# B&R Automation Studio project ACOPOStrak_DATech_Pilot (part 3)

### Config_1.assembly - 5PC900_TS17_00/mappMotion/TrakOval/Config_1.assembly
```
Element gAsmMain (Type=assembly)
  Tracks:
    TrackSeparation = 0.030
    Track[1]:
      Segments:
        SegmentRef[1] = ::Seg_A_1
        SegmentRef[2] = ::Seg_A_2
        SegmentRef[3] = ::Seg_A_3
        SegmentRef[4] = ::Seg_A_4
        SegmentRef[5] = ::Seg_A_5
        SegmentRef[6] = ::Seg_A_6
        SegmentRef[7] = ::Seg_A_7
        SegmentRef[8] = ::Seg_A_8
        SegmentRef[9] = ::Seg_A_9
        SegmentRef[10] = ::Seg_A_10
        SegmentRef[11] = ::Seg_A_11
        SegmentRef[12] = ::Seg_A_12
        SegmentRef[13] = ::Seg_A_13
        SegmentRef[14] = ::Seg_A_14
        SegmentRef[15] = ::Seg_A_15
        SegmentRef[16] = ::Seg_A_16
        SegmentRef[17] = ::Seg_A_17
        SegmentRef[18] = ::Seg_A_18
        SegmentRef[19] = ::Seg_A_19
        SegmentRef[20] = ::Seg_A_20
        SegmentRef[21] = ::Seg_A_21
        SegmentRef[22] = ::Seg_A_22
        SegmentRef[23] = ::Seg_A_23
        SegmentRef[24] = ::Seg_A_24
        SegmentRef[25] = ::Seg_A_25
        SegmentRef[26] = ::Seg_A_26
      Position = Absolute
        SegmentRef = ::Seg_A_11
        SegmentCountDirection = RightToLeft
        Position = 0
        Translation:
          X = 0.0
          Y = 0.0
          Z = 0.0
        Orientation:
          Angle1 = 0.0
          Angle2 = 0.0
          Angle3 = 180
  CommonSegmentSettings:
    SegmentSimulationOnPLC = Off
    ElongationCompensation = Inactive
    StopReaction = InductionHalt
    SpeedFilter = Lowpass
      FilterTime = 0.002
    ControllerParameters:
      DefaultParameter:
        Controller:
          Position:
            ProportionalGain = 220
          Speed:
            ProportionalGain = 60
            IntegrationTime = 0.0
          FeedForward:
            TotalMass = 1.8
            ForcePositive = 2
            ForceNegative = 2
            SpeedForceFactor = 2
            ForceLoad = 0.0
        MovementErrorLimits:
          PositionError = 1
          VelocityError = 100
      AdditionalParameterSets = NotUsed
    ScopeOfErrorReaction = Assembly
    ShuttleIdentificationTime = 2
  Shuttles:
    MaxShuttleCount = 50
    DistanceReserve:
      Collision = 0.002
      ErrorStop = 0.006
    ShuttleStereotypes:
      ShuttleStRef[1] = ShuttleStereotype_1
    MagnetPlateConfigurations:
      ShuttleType[1] = 8F1SA.203.xxxxxx-x
    CollisionAvoidance:
      Strategy = Constant
      MaximumModelDimensions:
        Length:
          ExtentToFront = 0.07
          ExtentToBack = 0.07
        Width:
          Width = 0.046
  AssemblyFeatures:
    AssemblyFeatureRef[1] = gSecLimit
    AssemblyFeatureRef[2] = Feature_Sim_Shuttle_Def
  Visualization:
    MonitoringPv = gShuttleMon
    ProcessingTaskClass = 1
```

### Config_2.shuttlestereotype - 5PC900_TS17_00/mappMotion/TrakOval/Config_2.shuttlestereotype
```
Element ShuttleStereotype_1 (Type=shuttlestereotype)
  MeasurementUnit = 5067858
  MeasurementResolution = 0.00001
  MovementLimits = Internal
    VelocityIsReadOnly = 0
    Velocity:
      Velocity = 2.5
    AccelerationIsReadOnly = 0
    Acceleration:
      Acceleration = 25
    DecelerationIsReadOnly = 0
    Deceleration:
      Deceleration = 25
    UpdateMode = Immediately
  JerkFilter = Used
    JerkTime = 0.02
  UserData:
    Size = 64
```

### Config_3.sector - 5PC900_TS17_00/mappMotion/TrakOval/Config_3.sector
```
Element SectorTrackA_1 (Type=sector)
  Type = Composed
    StartSegment:
      SegmentRef = ::Seg_A_24
    EndSegment:
      SegmentRef = ::Seg_A_25
      Position = 0
      PositionRelativeTo = FromEnd
Element SectorTrackA_2 (Type=sector)
  Type = Composed
    StartSegment:
      SegmentRef = ::Seg_A_3
    IntermediateSegments:
      SegmentRef[1] = ::Seg_A_4
      SegmentRef[2] = ::Seg_A_5
      SegmentRef[3] = ::Seg_A_6
    EndSegment:
      SegmentRef = ::Seg_A_7
      PositionRelativeTo = FromEnd
Element SectorTrackA_3 (Type=sector)
  Type = Composed
    StartSegment:
      SegmentRef = ::Seg_A_11
    EndSegment:
      SegmentRef = ::Seg_A_12
      PositionRelativeTo = FromEnd
Element SectorTrackA_4 (Type=sector)
  Type = Composed
    StartSegment:
      SegmentRef = ::Seg_A_16
    IntermediateSegments:
      SegmentRef[1] = ::Seg_A_17
      SegmentRef[2] = ::Seg_A_18
      SegmentRef[3] = ::Seg_A_19
    EndSegment:
      SegmentRef = ::Seg_A_20
      PositionRelativeTo = FromEnd
Element SectorTrackAll (Type=sector)
  Type = Composed
    StartSegment:
      SegmentRef = ::Seg_A_26
    IntermediateSegments:
      SegmentRef[1] = ::Seg_A_1
      SegmentRef[2] = ::Seg_A_2
      SegmentRef[3] = ::Seg_A_3
      SegmentRef[4] = ::Seg_A_4
      SegmentRef[5] = ::Seg_A_5
      SegmentRef[6] = ::Seg_A_6
      SegmentRef[7] = ::Seg_A_7
      SegmentRef[8] = ::Seg_A_8
      SegmentRef[9] = ::Seg_A_9
      SegmentRef[10] = ::Seg_A_10
      SegmentRef[11] = ::Seg_A_11
      SegmentRef[12] = ::Seg_A_12
      SegmentRef[13] = ::Seg_A_13
      SegmentRef[14] = ::Seg_A_14
      SegmentRef[15] = ::Seg_A_15
      SegmentRef[16] = ::Seg_A_16
      SegmentRef[17] = ::Seg_A_17
      SegmentRef[18] = ::Seg_A_18
      SegmentRef[19] = ::Seg_A_19
      SegmentRef[20] = ::Seg_A_20
      SegmentRef[21] = ::Seg_A_21
      SegmentRef[22] = ::Seg_A_22
      SegmentRef[23] = ::Seg_A_23
      SegmentRef[24] = ::Seg_A_24
    EndSegment:
      SegmentRef = ::Seg_A_25
      PositionRelativeTo = FromEnd
Element Sector3D (Type=sector)
  Type = Composed
    StartSegment:
      SegmentRef = ::Seg_A_19
      Position = 0.22
    EndSegment:
      SegmentRef = ::Seg_A_19
      Position = 0
      PositionRelativeTo = FromEnd
Element SectorCurve1 (Type=sector)
  Type = Composed
    StartSegment:
      SegmentRef = ::Seg_A_26
    IntermediateSegments:
      SegmentRef[1] = ::Seg_A_1
    EndSegment:
      SegmentRef = ::Seg_A_2
      PositionRelativeTo = FromEnd
Element SectorCurve2 (Type=sector)
  Type = Composed
    StartSegment:
      SegmentRef = ::Seg_A_19
    IntermediateSegments:
      SegmentRef[1] = 
    EndSegment:
      SegmentRef = ::Seg_A_19
      PositionRelativeTo = FromEnd
Element SectorCurve3 (Type=sector)
  Type = Composed
    StartSegment:
      SegmentRef = ::Seg_A_13
    IntermediateSegments:
      SegmentRef[1] = ::Seg_A_14
    EndSegment:
      SegmentRef = ::Seg_A_15
      PositionRelativeTo = FromEnd
Element SectorCurve4 (Type=sector)
  Type = Composed
    StartSegment:
      SegmentRef = ::Seg_A_21
    IntermediateSegments:
      SegmentRef[1] = ::Seg_A_22
    EndSegment:
      SegmentRef = ::Seg_A_23
      PositionRelativeTo = FromEnd
```

### Config_4.processpointlist - 5PC900_TS17_00/mappMotion/TrakOval/Config_4.processpointlist
```
Element ProcessPointList_1 (Type=processpointlist)
  ProcessPoint[0]:
    Name = ptCheckOut
    SectorRef = SectorTrackAll
    Position = 0.1
    PositionRelativeTo = FromEnd
    TriggerEventBufferSize = 10
    BarrierFunctionality = On
  ProcessPoint[1]:
    Name = ptCheckIn
    SectorRef = SectorTrackAll
    Position = 0.66
    PositionRelativeTo = FromEnd
    TriggerEventBufferSize = 30
    BarrierFunctionality = On
  ProcessPoint[2]:
    Name = pt3DIn
    SectorRef = SectorTrackAll
    Position = 10.52
    TriggerEventBufferSize = 10
    BarrierFunctionality = Off
  ProcessPoint[3]:
    Name = pt3DOut
    SectorRef = SectorTrackAll
    Position = 10.588
    PositionRelativeTo = FromEnd
    TriggerEventBufferSize = 10
    BarrierFunctionality = Off
  ProcessPoint[4]:
    Name = pt3D
    SectorRef = Sector3D
    TriggerEventBufferSize = 10
    BarrierFunctionality = Off
  ProcessPoint[5]:
    Name = ptCSZInt
    SectorRef = SectorTrackA_4
    Position = 1.76
    TriggerEventBufferSize = 10
    BarrierFunctionality = On
  ProcessPoint[6]:
    Name = ptCSZIn
    SectorRef = SectorTrackA_4
    Position = 1.75
    TriggerEventBufferSize = 10
    BarrierFunctionality = On
  ProcessPoint[7]:
    Name = ptCSZOut
    SectorRef = SectorTrackA_4
    Position = 2.02
    TriggerEventBufferSize = 10
    BarrierFunctionality = On
  ProcessPoint[8]:
    Name = ptUnloadingIn
    SectorRef = SectorCurve4
    Position = 0.76
    TriggerEventBufferSize = 10
    BarrierFunctionality = On
  ProcessPoint[9]:
    Name = ptUnloadingOut
    SectorRef = SectorCurve4
    Position = 0.88
    TriggerEventBufferSize = 10
    BarrierFunctionality = On
  ProcessPoint[10]:
    Name = ptVision
    SectorRef = SectorTrackAll
    Position = 7.1
    TriggerEventBufferSize = 10
    BarrierFunctionality = On
Element ProcessPointList_2 (Type=processpointlist)
  ProcessPoint[0]:
    Name = ptStage1
    SectorRef = SectorCurve1
    Position = 0.2295
    TriggerEventBufferSize = 10
    BarrierFunctionality = Off
  ProcessPoint[1]:
    Name = ptStage2
    SectorRef = SectorTrackA_2
    Position = 0.1778
    TriggerEventBufferSize = 10
    BarrierFunctionality = Off
  ProcessPoint[2]:
    Name = ptStage3
    SectorRef = SectorTrackA_2
    Position = 0.482
    TriggerEventBufferSize = 10
    BarrierFunctionality = Off
  ProcessPoint[3]:
    Name = ptStage4
    SectorRef = SectorTrackA_2
    Position = 0.715
    TriggerEventBufferSize = 10
    BarrierFunctionality = Off
  ProcessPoint[4]:
    Name = ptStage5
    SectorRef = SectorTrackA_2
    Position = 0.9375
    TriggerEventBufferSize = 10
    BarrierFunctionality = Off
  ProcessPoint[5]:
    Name = ptStage6
    SectorRef = SectorTrackA_2
    Position = 1.036
    TriggerEventBufferSize = 10
    BarrierFunctionality = Off
  ProcessPoint[6]:
    Name = ptStage7
    SectorRef = SectorTrackA_2
    Position = 2.231
    TriggerEventBufferSize = 10
    BarrierFunctionality = Off
  ProcessPoint[7]:
    Name = ptStage8
    SectorRef = SectorTrackA_2
    Position = 2.6712
    TriggerEventBufferSize = 10
    BarrierFunctionality = Off
  ProcessPoint[8]:
    Name = ptStage9
    SectorRef = SectorTrackA_2
    Position = 3.151
    TriggerEventBufferSize = 10
    BarrierFunctionality = Off
  ProcessPoint[9]:
    Name = ptStage10
    SectorRef = SectorTrackA_3
    Position = 0.801
    TriggerEventBufferSize = 10
    BarrierFunctionality = Off
  ProcessPoint[10]:
    Name = ptStage11
    SectorRef = SectorCurve3
    Position = 1.1005
    TriggerEventBufferSize = 10
    BarrierFunctionality = Off
  ProcessPoint[11]:
    Name = ptStage12
    SectorRef = SectorTrackA_4
    Position = 0.3805
    TriggerEventBufferSize = 10
    BarrierFunctionality = Off
  ProcessPoint[12]:
    Name = ptStage13
    SectorRef = SectorTrackA_4
    Position = 1.0407
    TriggerEventBufferSize = 10
    BarrierFunctionality = Off
  ProcessPoint[13]:
    Name = ptStage14
    SectorRef = SectorTrackA_4
    Position = 2.0096
    TriggerEventBufferSize = 10
    BarrierFunctionality = Off
  ProcessPoint[14]:
    Name = ptStage15
    SectorRef = SectorTrackA_4
    Position = 2.751
    TriggerEventBufferSize = 10
    BarrierFunctionality = Off
  ProcessPoint[15]:
    Name = ptStage16
    SectorRef = SectorTrackA_4
    Position = 2.8605
    TriggerEventBufferSize = 10
    BarrierFunctionality = Off
  ProcessPoint[16]:
    Name = ptStage17
    SectorRef = SectorCurve4
    Position = 0.121
    TriggerEventBufferSize = 10
    BarrierFunctionality = Off
  ProcessPoint[17]:
    Name = ptStage18
    SectorRef = SectorCurve4
    Position = 0.9179
    TriggerEventBufferSize = 10
    BarrierFunctionality = Off
  ProcessPoint[18]:
    Name = ptStage19
    SectorRef = SectorTrackA_1
    Position = 0.601
    TriggerEventBufferSize = 10
    BarrierFunctionality = Off
  ProcessPoint[19]:
    Name = ptBuffer
    SectorRef = SectorTrackAll
    Position = 0
    TriggerEventBufferSize = 10
    BarrierFunctionality = On
```

### Limits.assemblyfeature - 5PC900_TS17_00/mappMotion/TrakOval/Limits.assemblyfeature
```
Element gSecLimit (Type=assemblyfeature)
  Type = LocalLimits
    LocalLimit[1]:
      Location:
        SectorRef = Sector3D
      MotionLimits:
        Velocity = Basic
          Velocity = 0.25
```

### cfgAudit.mpaudittrail - 5PC900_TS17_00/mappServices/cfgAudit.mpaudittrail
```
Element gAuditTrak (Type=mpaudittrail)
  Audit:
    Events:
      [0] = 18
    RecordingSize = 16384
    SramBufferSize = 128
    TextSource = TXT
      OutputFormat = MpAudit/Event/Root
      Display = Ne
        Format = MpAudit/Event/RootDis
    Export:
      Encrypt = FALSE
  Alarms = None
```

### viCompCR.visioncomponent - 5PC900_TS17_00/mappVision/viCompCR.visioncomponent
```
Element gCameraCodeReading (Type=visioncomponent)
  VisionApplicationReference = ViAppCodeReading
```

## Logical view

Binary libraries used (declarations not repeated): operator, runtime, astime, AsIecCon, AsBrStr, standard, sys_lib, AsIODiag, McBase, McAcpTrak, McAxis, ViBase 5.15.0, AsZip, FileIO, AsARCfg, powerlnk, AsEPL, AsIO, CoTrace, MpAxis, MpBase, McAcpAx, MTTypes, MTBasics 2.00.0, MTData 2.00.0, MTFilter 2.00.0, brsystem, AsBrMath, AsMbTCP, MpAudit 5.15.0

### Global.typ - Global data types
```iecst
(**)

TYPE
	E_ASM_STATUS :
		(
		E_ASM_UNKNOWN := 0,
		E_ASM_OFF := 1,
		E_ASM_ON := 2,
		E_ASM_IDLE := 3,
		E_ASM_PROCESS := 4,
		E_ASM_ERRORSTOP := 5,
		E_ASM_MANUAL := 6,
		E_ASM_POWER_ON := 10,
		E_ASM_POWER_OFF := 20,
		E_ASM_INITIALIZATION := 30,
		E_ASM_RECOVERY := 31,
		E_ASM_RESET := 40,
		E_ASM_STOPPING := 50,
		E_ASM_EMS := 60,
		E_ASM_CLEAN := 70
		);
	E_PROCESS_STATUS :
		(
		E_PROCESS_None,
		E_PROCESS_Stage1,
		E_PROCESS_Stage2,
		E_PROCESS_Stage3,
		E_PROCESS_Stage4,
		E_PROCESS_Stage5,
		E_PROCESS_Stage6,
		E_PROCESS_Stage7,
		E_PROCESS_Stage8,
		E_PROCESS_Stage9,
		E_PROCESS_Stage10,
		E_PROCESS_Stage11,
		E_PROCESS_Stage12,
		E_PROCESS_Stage13,
		E_PROCESS_Stage14,
		E_PROCESS_Stage15,
		E_PROCESS_Stage16,
		E_PROCESS_Stage17,
		E_PROCESS_Stage18,
		E_PROCESS_Stage19
		);
END_TYPE

(**)

TYPE
	ShuttleUserData_typ : 	STRUCT
		SerialNumber : STRING[19]; (*Shuttle Number*)
		ProcessStatus : E_PROCESS_STATUS;
		Data : ARRAY[0..19]OF UINT;
	END_STRUCT;
END_TYPE

(**)

TYPE
	Command_type : 	STRUCT
		PowerOn : BOOL;
		PowerOff : BOOL;
		Initialize : BOOL;
		EMS : BOOL;
		Start : BOOL;
		Stop : BOOL;
		Reset : BOOL;
		ErrorReset : BOOL;
		Clean : BOOL;
	END_STRUCT;
	Parameter_type : 	STRUCT
		MovementPar : MovementParameter_type;
		PositionOffset : PosOffsetParameter_type;
		ProcessPosition : PositionParameter_type;
		TargetPPM : UINT := 30;
		CountOfGroup : USINT := 6;
	END_STRUCT;
	Status_type : 	STRUCT
		AsmState : E_ASM_STATUS;
	END_STRUCT;
END_TYPE

(**)

TYPE
	MovementParameter_type : 	STRUCT
		Initialize : SerializeParType;
		Stage1 : ServeStageParType;
		Stage2 : TransferStageParType;
		Stage3 : TransferStageParType;
		Stage4 : TransferStageParType;
		Stage5 : TransferStageParType;
		Stage6 : TransferStageParType;
		Stage7 : TransferStageParType;
		Stage8 : TransferStageParType;
		Stage9 : TransferStageParType;
		Stage10 : TransferStageParType;
		Stage11 : TransferStageParType;
		Stage12 : TransferStageParType;
		Stage13 : TransferStageParType;
		Stage14 : TransferStageParType;
		Stage15 : TransferStageParType;
		Stage16 : TransferStageParType;
		Stage17 : TransferStageParType;
		Stage18 : TransferStageParType;
		Stage19 : TransferStageParType;
		Return : SerializeParType;
	END_STRUCT;
	PositionParameter_type : 	STRUCT
		Stage : ARRAY[0..18]OF LREAL;
	END_STRUCT;
	PosOffsetParameter_type : 	STRUCT
		Stage : ARRAY[0..18]OF LREAL;
	END_STRUCT;
END_TYPE

(**)

TYPE
	ServeStageParType : 	STRUCT
		Velocity : REAL;
		Acceleration : REAL;
		Deceleration : REAL;
		MaxController : USINT;
	END_STRUCT;
	TransferStageParType : 	STRUCT
		Velocity : REAL;
		Acceleration : REAL;
		Deceleration : REAL;
		MaxController : USINT;
	END_STRUCT;
	SerializeParType : 	STRUCT
		RoutedVelocity : REAL;
		Velocity : REAL;
		Acceleration : REAL;
		Deceleration : REAL;
	END_STRUCT;
END_TYPE

(**)
```

### Global.var - Global variables
```iecst
VAR
	gShuttleMon : McAcpTrakAssemblyMonData;
END_VAR
(**)
VAR
	gLocal : BOOL;
	gManual : BOOL;
	gCmdRemote : Command_type;
	gCmd : Command_type;
END_VAR
VAR RETAIN
	gParInitialized : BOOL;
	gPar : Parameter_type;
END_VAR
VAR
	gSts : Status_type;
END_VAR
(**)
VAR
	gSim : BOOL;
END_VAR
(**)
VAR
	SIZE_OF_USERDATA : UDINT := 64; (*24*)
END_VAR
(*3D *)
VAR
	g3DStartPos : LREAL := 10.52;
	g3DEndPos : LREAL := 10.588;
END_VAR
(*Vision*)
VAR
	gShuttleTotalCount : DINT;
	gInitialDone : BOOL;
END_VAR
(*Barrier at buffer*)
VAR
	BrBuffer : MC_BR_BarrierCommand_AcpTrak;
END_VAR
```

### GlobalConst.var
```iecst
VAR CONSTANT
	ASM_MAX_TARGET : USINT := 20;
END_VAR
```

### Package Logical/Libraries - Global libraries

### Library Logical/Libraries/MyTrak (ANSIC)
Depends on: standard, AsBrStr, McAcpTrak, McAxis, McBase

#### Types.typ
```iecst
(**)
(*Enumeration*)

TYPE
	E_SLOT_IF_STATE :
		(
		E_SLOT_UNKNOWN := 0,
		E_SLOT_MANUAL := 1,
		E_SLOT_IDLE := 2,
		E_SLOT_PROCESS_READY := 3,
		E_SLOT_PROCESSING := 4,
		E_SLOT_TAKEOUT_READY := 5
		) := E_SLOT_UNKNOWN;
END_TYPE

(**)
(*Structure*)

TYPE
	MyTrakSlotType : 	STRUCT  (*Slot of Stage.*)
		Enable : BOOL;
		Sector : UDINT;
		Position : LREAL;
		Interface : E_SLOT_IF_STATE;
		Shuttle : McAxisType;
		NextStage : UDINT;
	END_STRUCT;
	MyTrakSlotTransType : 	STRUCT  (*Function Block for transfer Shuttle from Prestage to Nextstage*)
		moveAbs : MC_BR_RoutedMoveAbs_AcpTrak;
		axis : McAxisType;
		targetSlot : REFERENCE TO MyTrakSlotType;
		next : REFERENCE TO MyTrakSlotTransType;
	END_STRUCT;
	MyTrakSerializeType : 	STRUCT  (*Function Block for transfer Shuttle from Prestage to Nextstage*)
		moveVel : MC_BR_RoutedMoveVel_AcpTrak;
		axis : McAxisType;
		sourceSlot : REFERENCE TO MyTrakSlotType;
		next : REFERENCE TO MyTrakSerializeType;
	END_STRUCT;
END_TYPE

(**)
(*Internal Structrue for FunctionBlock*)

TYPE
	MyTrak_ServeStage_Internal_type : 	STRUCT
		slotMoveFc : REFERENCE TO MyTrakSlotTransType;
		fbTrgInfo : MC_BR_TrgPointGetInfo_AcpTrak;
		fbTrgEnable : MC_BR_TrgPointEnable_AcpTrak;
	END_STRUCT;
	MyTrak_TransStage_Internal_type : 	STRUCT
		slotMoveFc : REFERENCE TO MyTrakSlotTransType;
		manualCmd : R_TRIG;
	END_STRUCT;
	MyTrak_Serialize_Internal_type : 	STRUCT
		serialMoveFc : REFERENCE TO MyTrakSerializeType;
		manualCmd : R_TRIG;
	END_STRUCT;
	MyTrak_TicketArea_Internal_type : 	STRUCT
		step : USINT;
		init : BOOL;
		fbInEnable : MC_BR_TrgPointEnable_AcpTrak;
		fbInGetInfo : MC_BR_TrgPointGetInfo_AcpTrak;
		fbBarrierReadInfo : MC_BR_BarrierReadInfo_AcpTrak;
		fbBarrier : MC_BR_BarrierCommand_AcpTrak;
		fbOutEnable : MC_BR_TrgPointEnable_AcpTrak;
		fbOutGetInfo : MC_BR_TrgPointGetInfo_AcpTrak;
	END_STRUCT;
	MyTrak_ChangeVel_Internal_type : 	STRUCT
		step : DINT;
		preActive : BOOL;
		ElasticMoveVel : MC_BR_ElasticMoveVel_AcpTrak;
		TrgEnable : MC_BR_TrgPointEnable_AcpTrak;
		TrgGetInfo : MC_BR_TrgPointGetInfo_AcpTrak;
	END_STRUCT;
	MyTrak_ShInfeeder_Internal_type : 	STRUCT
		BarCmd : MC_BR_BarrierCommand_AcpTrak;
		BarReadInfo : MC_BR_BarrierReadInfo_AcpTrak;
		Tmr : TON;
		manualCmd : R_TRIG;
	END_STRUCT;
	MyTrak_Buffer_Internal_type : 	STRUCT
		slotMoveFc : REFERENCE TO MyTrakSlotTransType;
		CheckInPointEnable : MC_BR_TrgPointEnable_AcpTrak;
		GetCheckInShuttleInfo : MC_BR_TrgPointGetInfo_AcpTrak;
		GetShuttleInfo : MC_BR_ShReadInfo_AcpTrak;
		CheckOutBarrier : MC_BR_BarrierCommand_AcpTrak;
		Tmr : TON;
		manualCmd : R_TRIG;
		outReqCount : USINT;
	END_STRUCT;
	MyTrak_UntilStop_Internal_type : 	STRUCT
		serialMoveFc : REFERENCE TO MyTrakSerializeType;
		getShuttle : MC_BR_SecGetShuttleSel_AcpTrak;
	END_STRUCT;
END_TYPE
```

#### Constants.var
```iecst
(**)
VAR CONSTANT
	MyTrakIdle : DINT := 0;
	MyTrakRun : DINT := 1;
	MyTrakManual : DINT := 2;
	MyTrakNotEnoughShuttle : DINT := 40000;
	MyTrakMaximumControllerOverflow : DINT := 40001;
	MyTrakMinimumControllerUnderflow : DINT := 40002;
	MyTrakBusy : DINT := 65534;
	MyTrakDisabled : DINT := 65535;
END_VAR
(**)
VAR CONSTANT
	MyTrakNotExistSourceStage : DINT := -40000;
	MyTrakNotExistTargetStage : DINT := -40001;
	MyTrakNotExistSourceProcessPoint : DINT := -40002;
	MyTrakNotExistSourceCheckIn : DINT := -40003;
	MyTrakNotExistSourceCheckOut : DINT := -40004;
	MyTrakNotExistCheckinPt : DINT := -40000;
END_VAR
```

#### MyTrak.fun - Function and Function Block Define
```iecst
(**)
(*Function Blocks*)

{REDUND_ERROR} FUNCTION_BLOCK MyTrak_ShInfeeder (*Buffer Handle based Productivity *) (*$GROUP=User,$CAT=User,$GROUPICON=User.png,$CATICON=User.png*)
	VAR_INPUT
		Enable : BOOL; (*Enable/Disable*)
		ProcessPoint : REFERENCE TO McProcessPointType; (*Stop Position Process Point*)
		SetPPM : UINT; (*SettedPPM*)
		CountOfOneShot : USINT; (*Supply Shuttle Count at once*)
		Process : BOOL; (*Feeding Start/Stop*)
		Pause : BOOL; (*Puase when feeding is started*)
		Manual : BOOL; (*Manual Input when Feeding is Stopped - Positive Trigger*)
	END_VAR
	VAR_OUTPUT
		Active : BOOL; (*Activated FunctionBlock*)
		Error : BOOL; (*Error Status - Not Implemented*)
		ErrorID : DINT; (*Function Block Status - refer to Constant*)
		ActPPM : UINT; (*Actual PPM*)
		Interval : REAL; (*Feeding Interval*)
	END_VAR
	VAR
		Internal : MyTrak_ShInfeeder_Internal_type;
	END_VAR
END_FUNCTION_BLOCK

{REDUND_ERROR} FUNCTION_BLOCK MyTrak_Buffer (*Buffer Handing based Productivity*) (*$GROUP=User,$CAT=User,$GROUPICON=User.png,$CATICON=User.png*)
	VAR_INPUT
		Enable : BOOL; (*Activate Function Block*)
		CheckInProcessPoint : REFERENCE TO McProcessPointType; (*Check In Process Point*)
		CheckOutProcessPoint : REFERENCE TO McProcessPointType; (*Check Out Process Point*)
		TargetStage : UDINT; (*Reference of Target Stage(MyTrakSlotType array)*)
		TargetSlotCount : USINT; (*Count of slot in target stage*)
		Process : BOOL; (*Process Start And Stop*)
		Feeding : BOOL; (*Holding Process*)
		Manual : BOOL; (*Manual Feeding*)
		SetPPM : UINT; (*Set PPM*)
		CountOfOneShot : USINT; (*Feeding Shuttle Count of One Time*)
		MaximumShuttleCount : USINT; (*Maximum Handle Shuttle Count*)
		Velocity : REAL; (*Velocity from Buffer to 'Target Stage'*)
		Acceleration : REAL; (*Acceleration from Buffer to 'Target Stage'*)
		Deceleration : REAL; (*Deceleration from Buffer to 'Target Stage'*)
		AdvancedParameters : McAcpTrakAdvRouteParType; (*Advanced Parameter*)
	END_VAR
	VAR_OUTPUT
		Active : BOOL; (*Activate Status*)
		Error : BOOL; (*Error Status*)
		ErrorID : DINT; (*Error ID*)
		CountOfShuttle : USINT; (*Total Shuttle by Handled By this FunctionBlock*)
		CountOfBuffer : USINT; (*Shuttle Count in Buffer*)
		CountOfSupplied : UDINT; (*Shuttle Count in Buffer*)
		NextSlotNo : INT; (*Next Slot Number*)
		Interval : REAL; (*Feeding Interval*)
	END_VAR
	VAR
		Internal : MyTrak_Buffer_Internal_type;
	END_VAR
END_FUNCTION_BLOCK

{REDUND_ERROR} FUNCTION_BLOCK MyTrak_ServeStage (*Move shuttles  from source process point to stage*) (*$GROUP=User,$CAT=User,$GROUPICON=User.png,$CATICON=User.png*)
	VAR_INPUT
		Enable : BOOL; (*Activate Function Block*)
		SourceProcessPoint : REFERENCE TO McProcessPointType; (*Reference of Process Point that shuttle getting*)
		TargetStage : UDINT; (*Reference of Target Stage(MyTrakSlotType array)*)
		TargetSlotCount : USINT; (*Count of slot in target stage*)
		MaximumShuttleCount : USINT; (*Maximum Handle Shuttle Count*)
		MinimumShuttleCount : USINT; (*Minimum Shuttle Handle Count at one time*)
		Velocity : REAL; (*Velocity from 'Source Stage' to 'Target Stage'.*)
		Acceleration : REAL; (*Acceleration from Source Process Point*)
		Deceleration : REAL; (*Deceleration from Source Process Point *)
		AdvancedParameters : McAcpTrakAdvRouteParType; (*Advanced Parameter*)
	END_VAR
	VAR_OUTPUT
		Active : BOOL; (*Activate Status*)
		Error : BOOL; (*Error Status*)
		ErrorID : DINT; (*Error ID*)
		CountOfShuttle : INT; (*Count of Shuttles*)
		NextSlotNo : INT; (*Next Placed Slot*)
	END_VAR
	VAR
		Internal : MyTrak_ServeStage_Internal_type;
	END_VAR
END_FUNCTION_BLOCK

{REDUND_ERROR} FUNCTION_BLOCK MyTrak_TransStage (*Move shuttles from source stage to target stage *) (*$GROUP=User,$CAT=User,$GROUPICON=User.png,$CATICON=User.png*)
	VAR_INPUT
		Enable : BOOL; (*Activate Function Block*)
		SourceStage : {REDUND_UNREPLICABLE} ARRAY[0..9] OF UDINT; (*Reference of Source Stage(Reference of 'MyTrakSlotType' array)*)
		SourceSlotCount : {REDUND_UNREPLICABLE} ARRAY[0..9] OF USINT; (*Source Stage Slot Count*)
		TargetStage : {REDUND_UNREPLICABLE} UDINT; (*Reference of Target Stage(Reference of 'MyTrakSlotType' array)*)
		TargetSlotCount : USINT; (*Target Stage Slot Count*)
		MaximumShuttleCount : USINT; (*Maximum Shuttle Count between 'End of Source Slot' to 'End of Target Slot')*)
		Process : BOOL; (*Transfer Start / Stop*)
		Manual : BOOL; (*Manual Feeding One Shuttle(By Positive Edge)*)
		Velocity : REAL; (*Velocity from 'Source Stage' to 'Target Stage'.*)
		Acceleration : REAL; (*Acceleration from 'Source Stage' to 'Target Stage'.*)
		Deceleration : REAL; (*Deceleration from 'Source Stage' to 'Target Stage'*)
		AdvancedParameters : McAcpTrakAdvRouteParType; (*Advanced Parameter for Make Routing - Refer *)
	END_VAR
	VAR_OUTPUT
		Active : BOOL; (*Activate Status*)
		Error : BOOL; (*Error Status*)
		ErrorID : DINT; (*Error ID*)
		CountOfShuttle : INT; (*Count of Shuttles*)
		NextSlotNo : INT; (*Next Placed Slot*)
	END_VAR
	VAR
		Internal : MyTrak_TransStage_Internal_type;
	END_VAR
END_FUNCTION_BLOCK

{REDUND_ERROR} FUNCTION_BLOCK MyTrak_Serialize (*Move shuttles from source stage to target sector*) (*$GROUP=User,$CAT=User,$GROUPICON=User.png,$CATICON=User.png*)
	VAR_INPUT
		Enable : BOOL; (*Activate Function Block*)
		SourceStage : ARRAY[0..9] OF UDINT; (*Reference of Source Stage(Reference of MyTrakSlotType array)*)
		SourceSlotCount : ARRAY[0..9] OF USINT; (*Source Array Count*)
		TargetSector : REFERENCE TO McSectorType; (*Reference of Target Sector(Reference of McSectorType)*)
		TargetPosition : LREAL; (*Target Sector Position*)
		Process : BOOL; (*Serialize Start / Stop*)
		Manual : BOOL; (*Manual Feeding One Shuttle(By Positive Edge)*)
		RoutedVelocity : REAL; (*Routed Velocity from Stage to Target Position*)
		Velocity : REAL; (*Velocty from Target Position Of Sector*)
		Acceleration : REAL; (*Acceleration*)
		Deceleration : REAL; (*Deceleration*)
		AdvancedParameters : McAcpTrakAdvRouteParType; (*Advanced Parameter for moving*)
	END_VAR
	VAR_OUTPUT
		Active : BOOL; (*Activate Status*)
		Error : BOOL; (*Error Status*)
		ErrorID : DINT; (*Error ID or Status ID*)
		CountOfShuttle : INT; (*Count of shuttle by handled by this FunctionBlock*)
	END_VAR
	VAR
		Internal : MyTrak_Serialize_Internal_type;
	END_VAR
END_FUNCTION_BLOCK

{REDUND_ERROR} FUNCTION_BLOCK MyTrak_UntilStop (*Not Implemented*) (*$GROUP=User,$CAT=User,$GROUPICON=User.png,$CATICON=User.png*)
	VAR_INPUT
		SourceSector : REFERENCE TO McSectorType;
		SourceStart : LREAL;
		SourceEnd : LREAL;
		Execute : REAL;
		TargetSector : REFERENCE TO McSectorType;
		TargetPosition : REAL;
		RoutedVelocity : REAL;
		Velocity : REAL;
		Acceleration : REAL;
		Deceleration : REAL;
		AdvancedParameters : McAcpTrakAdvRouteParType;
	END_VAR
	VAR_OUTPUT
		Active : BOOL;
		Error : BOOL;
		ErrorID : DINT;
		Done : BOOL;
		CountOfShuttle : INT;
	END_VAR
	VAR
		Internal : MyTrak_UntilStop_Internal_type;
	END_VAR
END_FUNCTION_BLOCK

{REDUND_ERROR} FUNCTION_BLOCK MyTrak_TicketArea (*Keep shuttles count between two process point*) (*$GROUP=User,$CAT=User,$GROUPICON=User.png,$CATICON=User.png*)
	VAR_INPUT
		Enable : BOOL; (*Activating Function Block*)
		InPoint : REFERENCE TO McProcessPointType; (*Start Point*)
		OutPoint : REFERENCE TO McProcessPointType; (*End Point*)
		MaximumShuttleCount : USINT; (*Keeping Shuttle Count*)
		InitShuttleCount : USINT; (*Initial Shuttle Count(It means shuttle count of prcess In to Process Out before activatiing*)
	END_VAR
	VAR_OUTPUT
		Active : BOOL; (*Activate Status*)
		Error : BOOL; (*Error Status*)
		ErrorID : DINT; (*Status ID*)
		Processing : BOOL;
		Passed : BOOL;
		ShuttleCount : USINT;
	END_VAR
	VAR
		Internal : {REDUND_UNREPLICABLE} MyTrak_TicketArea_Internal_type;
	END_VAR
END_FUNCTION_BLOCK

{REDUND_ERROR} FUNCTION_BLOCK MyTrak_ChangeVel (*Change Shuttle Velocity at Specific Process Point*) (*$GROUP=User,$CAT=User,$GROUPICON=User.png,$CATICON=User.png*)
	VAR_INPUT
		Enable : BOOL; (*Enable*)
		ProcessPoint : REFERENCE TO McProcessPointType;
		Velocity : REAL; (*Changing Velocity*)
		Acceleration : REAL; (*Changing Acceleration*)
		Deceleration : {REDUND_UNREPLICABLE} REAL; (*Chagneing Deceleration*)
		Direction : {REDUND_UNREPLICABLE} McDirectionEnum; (*Changing Direction*)
	END_VAR
	VAR_OUTPUT
		Active : BOOL; (*Enable Status*)
		Error : BOOL; (*Error Existing*)
		ErrorID : DINT; (*Error ID*)
	END_VAR
	VAR
		Internal : MyTrak_ChangeVel_Internal_type; (*Internal Variable*)
	END_VAR
END_FUNCTION_BLOCK
(**)
(*Functions*)

{REDUND_ERROR} FUNCTION GetProcessReady : BOOL (*All Stage Process Ready Status*) (*$GROUP=User,$CAT=User,$GROUPICON=User.png,$CATICON=User.png*)
	VAR_INPUT
		Stage : UDINT;
		SlotCount : USINT;
	END_VAR
END_FUNCTION

{REDUND_ERROR} FUNCTION GetProcessing : BOOL (*All Stage Processing Status*) (*$GROUP=User,$CAT=User,$GROUPICON=User.png,$CATICON=User.png*)
	VAR_INPUT
		Stage : UDINT;
		SlotCount : USINT;
	END_VAR
END_FUNCTION

{REDUND_ERROR} FUNCTION GetStageStatus : E_SLOT_IF_STATE (*All Stage Process Ready Status*) (*$GROUP=User,$CAT=User,$GROUPICON=User.png,$CATICON=User.png*)
	VAR_INPUT
		Stage : UDINT;
		SlotCount : USINT;
	END_VAR
END_FUNCTION

{REDUND_ERROR} FUNCTION InitializeFcBank : BOOL (*Initialize Maximum Movement FunctionBlock Count*) (*$GROUP=User,$CAT=User,$GROUPICON=User.png,$CATICON=User.png*)
	VAR_INPUT
		shuttleCount : UINT;
	END_VAR
END_FUNCTION

{REDUND_ERROR} FUNCTION Random : BOOL (*Get RandomValue in Boolean*) (*$GROUP=User,$CAT=User,$GROUPICON=User.png,$CATICON=User.png*)
	VAR_INPUT
		Percent : REAL; (*Percent of return 'TRUE'*)
	END_VAR
END_FUNCTION
```

#### MyTrakFunc.h - Additional Header for all function
```c
//Rent MyTrakSlotTransTyoe from Back
MyTrakSlotTransType* rentRoutedAbsFc();

//Rent and Attach MyTrakSerializeType from Back
MyTrakSlotTransType* attachRoutedAbsFc(MyTrakSlotTransType** rootSlotMove);

//Return MyTrakSlotTransTyoe from Back
void rtnRoutedAbsFc(MyTrakSlotTransType* rtnFc);

//Rent MyTrakSerializeType from Back
MyTrakSerializeType* rentRoutedVelFc();

//Rent and Attach MyTrakSerializeType from Back
MyTrakSerializeType* attachRoutedVelFc(MyTrakSerializeType** rootSerialize);

//Return MyTrakSerializeType to Back
void rtnRoutedVelFc(MyTrakSerializeType* rtnFc);

//Search Next slot of stage
int SearchNextSlot(UDINT firstSlot, int currentSlot, unsigned int slotCount);

//Realease list of MyTrakSlotTransType
void releaseMyTrakSlotTran(MyTrakSlotTransType** executeList);

//Realease list of MyTrakSerializeType
void releaseMyTrakSerialize(MyTrakSerializeType** executeList);

//execute list of MyTrakSlotTransType
DINT execMyTrakSlotTrans(MyTrakSlotTransType** executeList);

//execute list of MyTrakSerializeType
DINT execMyTrakSerialize(MyTrakSerializeType** executeList);
```

#### MyTrak_Buffer.c - Shuttle Feeding System
```c
/********************************************************************
 * COPYRIGHT -- B&R Korea
 ********************************************************************
 * File: MyTrak_Buffer.c
 * Author: Taeryoung Ok
 * Created: 2021/11/06
 ********************************************************************
 * Description: Manager Buffer Area for Trak System
 ********************************************************************/

#include <bur/plctypes.h>
#ifdef __cplusplus
	extern "C"
	{
#endif
	#include "MyTrak.h"
	#include "MyTrakFunc.h"
#ifdef __cplusplus
	};
#endif

#define NULL 0
#define FALSE 0
#define TRUE 1

/* Buffer System */
void MyTrak_Buffer(struct MyTrak_Buffer* inst)
{
	int loop = 0, unuseableSlotCount = 0;

	MyTrakSlotType* slot;

	MyTrakSlotTransType* 	newSlotMove;

	if (inst->Enable == TRUE && inst->Active == FALSE)
	{	//Disabled -> Enable
		inst->Internal.CheckInPointEnable.Enable 	= TRUE;
		inst->Internal.CheckOutBarrier.Execute 		= TRUE;
		inst->Internal.CheckOutBarrier.Command 		= mcACPTRAK_BARRIER_CLOSE;
		inst->CountOfSupplied 						= 0;

		if (inst->Internal.CheckInPointEnable.Valid == TRUE && inst->Internal.CheckOutBarrier.Done == TRUE)
		{
			inst->Active = TRUE;
		}
	}
	else if (inst->Enable == FALSE && inst->Active == TRUE)
	{	//Enable ->Disable
		inst->Internal.CheckInPointEnable.Enable 	= FALSE;
		inst->Internal.GetShuttleInfo.Enable		= FALSE;
		inst->Internal.GetCheckInShuttleInfo.Execute= FALSE;
		inst->Internal.CheckOutBarrier.Execute 		= TRUE;
		inst->Internal.CheckOutBarrier.Command 		= mcACPTRAK_BARRIER_OPEN;
		inst->Internal.GetShuttleInfo.Enable		= FALSE;
		inst->Internal.outReqCount					= 0;

		if (inst->Internal.CheckInPointEnable.Valid == FALSE && inst->Internal.CheckOutBarrier.Done == TRUE)
		{
			releaseMyTrakSlotTran(&inst->Internal.slotMoveFc);

			for (loop = 0; loop < inst->TargetSlotCount; loop++)
			{
				slot 			= (MyTrakSlotType*)(inst->TargetStage + sizeof(MyTrakSlotType) * loop);
				brsmemset((UDINT)&slot->Shuttle, 0, sizeof(McAxisType));
				slot->Interface = E_SLOT_UNKNOWN;
			}
			inst->Active = FALSE;
		}
	}
	else if (inst->Enable == TRUE && inst->Active == TRUE)
	{
		//Error Check

		//Shuttle Count Check in Target Stage
		for (loop = 0; loop < inst->TargetSlotCount; loop++)
		{
			slot = (MyTrakSlotType*)(inst->TargetStage + sizeof(MyTrakSlotType) * loop);

			if (slot->Shuttle.controlif != 0)
				unuseableSlotCount++;
		}

		//Add Request Count of Buffer
		if (inst->Process == TRUE)
		{
			// Auto Mode Handle
			if (inst->Feeding == FALSE)
			{
				inst->ErrorID = MyTrakIdle;
			}
			else
			{
				if (inst->Internal.Tmr.Q == TRUE)
				{
					if (inst->CountOfShuttle + unuseableSlotCount >= inst->MaximumShuttleCount)
					{	//Checking Max Controller Setting
						inst->ErrorID = MyTrakMaximumControllerOverflow;
					}
					else if ((inst->Internal.outReqCount + inst->CountOfOneShot) > inst->Internal.CheckInPointEnable.EventCount)
					{	//Checking Shuttle Count in Buffer
						inst->ErrorID = MyTrakNotEnoughShuttle;
					}
					else
					{
						inst->Internal.Tmr.IN 			= FALSE;
						inst->Internal.outReqCount		= inst->Internal.outReqCount + inst->CountOfOneShot;
						inst->ErrorID 					= MyTrakRun;
					}
				}
				else
				{
					//Resetarting Timer
					inst->Interval 						= 60000.0 / ((float)inst->SetPPM / (float)inst->CountOfOneShot);

					inst->Internal.Tmr.IN 				= TRUE;
					inst->Internal.Tmr.PT 				= inst->Interval;
					inst->ErrorID 						= MyTrakRun;
				}
			}
		}
		else
		{	//Manual Mode Handle
			inst->ErrorID = MyTrakManual;

			if (inst->Internal.manualCmd.Q == TRUE &&
				inst->Internal.CheckInPointEnable.EventCount > 0)
			{
				if (inst->CountOfShuttle + unuseableSlotCount >= inst->MaximumShuttleCount)
				{	//Checking Max Controller Setting
					inst->ErrorID = MyTrakMaximumControllerOverflow;
				}
				else if ((inst->Internal.outReqCount + inst->CountOfOneShot) > inst->Internal.CheckInPointEnable.EventCount)
				{	//Checking Shuttle Count in Buffer
					inst->ErrorID = MyTrakNotEnoughShuttle;
				}
				else
				{
					//Manual Operating
					inst->Internal.outReqCount = 1;
				}
			}
		}

		if (inst->Internal.outReqCount > 0 && inst->Internal.CheckInPointEnable.EventCount > 0)
			inst->Internal.GetCheckInShuttleInfo.Execute = TRUE;

		if (inst->Internal.GetCheckInShuttleInfo.Done == TRUE)
		{
			inst->Internal.GetShuttleInfo.Axis = &inst->Internal.GetCheckInShuttleInfo.TrgPointInfo.Axis;
			inst->Internal.GetShuttleInfo.Enable = TRUE;

			if (inst->Internal.GetShuttleInfo.Valid == TRUE)
			{
				if (inst->Internal.GetShuttleInfo.ShuttleInfo.AdditionalInfo.PLCopenState == mcAXIS_CONTINUOUS_MOTION)
				{
					//Select Target Slot
					if ((inst->NextSlotNo = SearchNextSlot(inst->TargetStage, inst->NextSlotNo, inst->TargetSlotCount)) != -1)
					{
						slot = (MyTrakSlotType*)(inst->TargetStage + sizeof(MyTrakSlotType) * inst->NextSlotNo);

						//Get New Last Slot Transfer Structure From FcBank
						newSlotMove = attachRoutedAbsFc(&inst->Internal.slotMoveFc);

						//Set Command Parameters
						newSlotMove->axis 					= inst->Internal.GetCheckInShuttleInfo.TrgPointInfo.Axis;
						newSlotMove->targetSlot 			= slot;

						newSlotMove->moveAbs.Axis			= &newSlotMove->axis;
						newSlotMove->moveAbs.Sector	 		= (McSectorType*)(newSlotMove->targetSlot->Sector);
						newSlotMove->moveAbs.Position	 	= newSlotMove->targetSlot->Position;
						newSlotMove->moveAbs.Velocity 		= inst->Velocity;
						newSlotMove->moveAbs.Acceleration 	= inst->Acceleration;
						newSlotMove->moveAbs.Deceleration 	= inst->Deceleration;
						newSlotMove->moveAbs.AdvancedParameters = inst->AdvancedParameters;

						newSlotMove->moveAbs.Execute 		= TRUE;

						//Add Ticket
						inst->Internal.CheckOutBarrier.AdvancedParameters.TicketCount = 1;
						inst->Internal.CheckOutBarrier.Command = mcACPTRAK_BARRIER_ADD_TICKETS;
						inst->Internal.CheckOutBarrier.Execute = TRUE;

						//Out Request Count
						inst->Internal.outReqCount--;
						inst->CountOfSupplied++;

						//Off Shuttle Info
						inst->Internal.GetCheckInShuttleInfo.Execute 					= FALSE;
						inst->Internal.GetShuttleInfo.Enable 							= FALSE;
					}
				}
				else
				{
					//Add Ticket
					inst->Internal.CheckOutBarrier.AdvancedParameters.TicketCount = 1;
					inst->Internal.CheckOutBarrier.Command = mcACPTRAK_BARRIER_ADD_TICKETS;
					inst->Internal.CheckOutBarrier.Execute = TRUE;

					//Off Shuttle Info
					inst->Internal.GetCheckInShuttleInfo.Execute 					= FALSE;
					inst->Internal.GetShuttleInfo.Enable 							= FALSE;
				}
			}
		}

		inst->CountOfBuffer = inst->Internal.CheckInPointEnable.EventCount;
		inst->CountOfShuttle = execMyTrakSlotTrans(&inst->Internal.slotMoveFc);
	}
	else if (inst->Enable == FALSE && inst->Active == FALSE)
	{	//Disabled
		releaseMyTrakSlotTran(&inst->Internal.slotMoveFc);
		inst->ErrorID = MyTrakDisabled;
	}

	inst->Internal.manualCmd.CLK = inst->Manual;
	R_TRIG(&inst->Internal.manualCmd);

	TON(&inst->Internal.Tmr);

	if (inst->Internal.CheckOutBarrier.Done == TRUE)
		inst->Internal.CheckOutBarrier.Execute = FALSE;

	//Exection Function Blocks
	inst->Internal.CheckInPointEnable.ProcessPoint = inst->CheckInProcessPoint;
	inst->Internal.GetCheckInShuttleInfo.ProcessPoint = inst->CheckInProcessPoint;
	inst->Internal.CheckOutBarrier.ProcessPoint = inst->CheckOutProcessPoint;

	MC_BR_TrgPointEnable_AcpTrak(&inst->Internal.CheckInPointEnable);
	MC_BR_TrgPointGetInfo_AcpTrak(&inst->Internal.GetCheckInShuttleInfo);
	MC_BR_ShReadInfo_AcpTrak(&inst->Internal.GetShuttleInfo);
	MC_BR_BarrierCommand_AcpTrak(&inst->Internal.CheckOutBarrier);
}
```

#### MyTrak_ServeStage.c - Move shuttles  from source process point to stage
```c
/********************************************************************
 * COPYRIGHT -- B&R Korea
 ********************************************************************
 * File: MyTrak_ServeStage.c
 * Author: Taeryoung Ok
 * Created: 2021/11/06
 ********************************************************************
 * Description: Serve Shuttle to Slot that is pass Source Process Point
 ********************************************************************/

#include <bur/plctypes.h>
#ifdef __cplusplus
	extern "C"
	{
#endif
	#include "MyTrak.h"
	#include "MyTrakFunc.h"
#ifdef __cplusplus
	};
#endif

#define NULL
#define FALSE 0
#define TRUE 1

void MyTrak_ServeStage(struct MyTrak_ServeStage* inst)
{
	int loop = 0, unuseableSlotCount = 0;
	MyTrakSlotType* 		slot;

	MyTrakSlotTransType* 	newSlotMove;

	//////////////////////////////////////////////////////////////////////
	if (inst->Enable == TRUE && inst->Active == FALSE)
	{
		inst->Internal.fbTrgEnable.Enable 	= TRUE;

		if (inst->Internal.fbTrgEnable.Valid == TRUE)
			inst->Active = TRUE;
	}
	else if (inst->Enable == FALSE && inst->Active == TRUE)
	{
		inst->Active 						= FALSE;
		inst->CountOfShuttle 				= 0;
		inst->NextSlotNo 					= 0;
		inst->Internal.fbTrgEnable.Enable 	= FALSE;

		releaseMyTrakSlotTran(&inst->Internal.slotMoveFc);

		for (loop = 0; loop < inst->TargetSlotCount; loop++)
		{
			slot 			= (MyTrakSlotType*)(inst->TargetStage + sizeof(MyTrakSlotType) * loop);
			brsmemset((UDINT)&slot->Shuttle, 0, sizeof(McAxisType));
			slot->Interface = E_SLOT_UNKNOWN;
		}
	}
	else if (inst->Enable == TRUE && inst->Active == TRUE)
	{
		//Trig Point Check

		//Slot Setting Check(Target Sector, Target Slot)

		//Shuttle Count Check in Target Stage
		for (loop = 0; loop < inst->TargetSlotCount; loop++)
		{
			slot = (MyTrakSlotType*)(inst->TargetStage + sizeof(MyTrakSlotType) * loop);

			if (slot->Shuttle.controlif != 0)
				unuseableSlotCount++;
		}

		//Shuttle Check
		if (inst->Internal.fbTrgEnable.EventCount > 0)
		{
			if (inst->CountOfShuttle + unuseableSlotCount >= inst->MaximumShuttleCount)
			{
				inst->ErrorID = MyTrakMaximumControllerOverflow;
			}
			else if ((inst->MinimumShuttleCount != 0 && inst->Internal.fbTrgEnable.EventCount + inst->CountOfShuttle < inst->MinimumShuttleCount))
			{
				inst->ErrorID = MyTrakMinimumControllerUnderflow;
			}
			else
			{
				inst->Internal.fbTrgInfo.Execute = TRUE;

				if ((inst->Internal.fbTrgInfo.Done == TRUE)
					&& ((inst->NextSlotNo = SearchNextSlot(inst->TargetStage, inst->NextSlotNo, inst->TargetSlotCount)) != -1))
				{
					slot = (MyTrakSlotType*)(inst->TargetStage + sizeof(MyTrakSlotType) * inst->NextSlotNo);

					//Get New Last Slot Transfer Structure From FcBank
					newSlotMove = attachRoutedAbsFc(&inst->Internal.slotMoveFc);

					//Set Command Parameters
					newSlotMove->axis 					= inst->Internal.fbTrgInfo.TrgPointInfo.Axis;
					newSlotMove->targetSlot 			= slot;

					newSlotMove->moveAbs.Axis	 		= &newSlotMove->axis;
					newSlotMove->moveAbs.Sector	 		= (McSectorType*)(newSlotMove->targetSlot->Sector);
					newSlotMove->moveAbs.Position	 	= newSlotMove->targetSlot->Position;
					newSlotMove->moveAbs.Velocity 		= inst->Velocity;
					newSlotMove->moveAbs.Acceleration 	= inst->Acceleration;
					newSlotMove->moveAbs.Deceleration 	= inst->Deceleration;
					newSlotMove->moveAbs.AdvancedParameters = inst->AdvancedParameters;

					newSlotMove->moveAbs.Execute 		= TRUE;

					inst->Internal.fbTrgInfo.Execute 	= FALSE;
				}

				if (inst->CountOfShuttle > 0)
					inst->ErrorID = MyTrakRun;
				else
					inst->ErrorID = MyTrakIdle;
			}
		}
		else
		{
			if (inst->CountOfShuttle > 0)
				inst->ErrorID = MyTrakRun;
			else
				inst->ErrorID = MyTrakIdle;
		}

		inst->CountOfShuttle = execMyTrakSlotTrans(&inst->Internal.slotMoveFc);
	}
	else if (inst->Enable == FALSE && inst->Active == FALSE)
	{
		releaseMyTrakSlotTran(&inst->Internal.slotMoveFc);
		inst->ErrorID = MyTrakDisabled;
	}

	//Execute Trigger Point FunctionBlocks
	inst->Internal.fbTrgEnable.ProcessPoint 	= inst->SourceProcessPoint;
	inst->Internal.fbTrgInfo.ProcessPoint 		= inst->SourceProcessPoint;

	MC_BR_TrgPointEnable_AcpTrak(&inst->Internal.fbTrgEnable);
	MC_BR_TrgPointGetInfo_AcpTrak(&inst->Internal.fbTrgInfo);
}
```

#### MyTrak_TransStage.c - Move shuttles from source stage to target stage 
```c
/********************************************************************
 * COPYRIGHT -- B&R Korea
 ********************************************************************
 * File: MyTrak_TransStage.c
 * Author: Taeryoung Ok
 * Created: 2021/11/06
 ********************************************************************
 * Description: Transfer Shuttle from Source stage to Target Stage
 ********************************************************************/

#include <bur/plctypes.h>
#ifdef __cplusplus
	extern "C"
	{
#endif
#include "MyTrak.h"
#include "MyTrakFunc.h"
#ifdef __cplusplus
	};
#endif

#define NULL 0
#define FALSE 0
#define TRUE 1

void MyTrak_TransStage(struct MyTrak_TransStage* inst)
{
	int 					preloop = 0, loop = 0, prestage = 0, unuseableSlotCount = 0;

	MyTrakSlotType* 		slot;
	MyTrakSlotType*			preslot;
	MyTrakSlotTransType*	newSlotMove;

	if (inst->Enable == TRUE && inst->Active == FALSE)
	{ //Disabled -> Enable
		inst->Active 		= TRUE;
	}
	else if (inst->Enable == FALSE && inst->Active == TRUE)
	{ //Enabled -> Disable
		inst->Active 		= FALSE;
		inst->ErrorID = MyTrakDisabled;
		inst->CountOfShuttle = 0;
		inst->NextSlotNo = 0;
		inst->Internal.manualCmd.CLK = FALSE; R_TRIG(&inst->Internal.manualCmd);

		releaseMyTrakSlotTran(&inst->Internal.slotMoveFc);

		for (loop = 0; loop < inst->TargetSlotCount; loop++)
		{
			slot 			= (MyTrakSlotType*)(inst->TargetStage + sizeof(MyTrakSlotType) * loop);
			brsmemset((UDINT)&slot->Shuttle, 0, sizeof(McAxisType));
			slot->Interface = E_SLOT_UNKNOWN;
		}
	}
	else if (inst->Enable == TRUE && inst->Active == TRUE)
	{ //Enabled
		//Manual Command Checking
		inst->Internal.manualCmd.CLK = inst->Manual; R_TRIG(&inst->Internal.manualCmd);

		if (inst->Process == TRUE || inst->Internal.manualCmd.Q)
		{
			//Slot Setting Check(Target Sector, Target Slot)

			//Shuttle Count Check in Target Stage
			for (loop = 0; loop < inst->TargetSlotCount; loop++)
			{
				slot = (MyTrakSlotType*)(inst->TargetStage + sizeof(MyTrakSlotType) * loop);

				if (slot->Shuttle.controlif != 0)
					unuseableSlotCount++;
			}

			for (prestage = 0; prestage < 10; prestage++)
			{
				for (preloop = inst->SourceSlotCount[prestage] - 1; preloop >= 0; preloop--)
				{
					//Source Slot Check
					preslot = (MyTrakSlotType*)(inst->SourceStage[prestage] + sizeof(MyTrakSlotType) * preloop);

					if ((preslot->Interface == E_SLOT_TAKEOUT_READY ||
						(preslot->Interface == E_SLOT_MANUAL && preslot->Shuttle.controlif != 0))
						&& preslot->NextStage == inst->TargetStage)
					{
						if (inst->CountOfShuttle + unuseableSlotCount >= inst->MaximumShuttleCount)
						{
							inst->ErrorID = MyTrakMaximumControllerOverflow;
						}
						else
						{
							inst->ErrorID = MyTrakBusy;

							//Select Target Slot
							if ((inst->NextSlotNo = SearchNextSlot(inst->TargetStage, inst->NextSlotNo, inst->TargetSlotCount)) == -1)
								break;
							else
								slot = (MyTrakSlotType*)(inst->TargetStage + sizeof(MyTrakSlotType) * inst->NextSlotNo);

							//Get New Last Slot Transfer Structure From FcBank
							newSlotMove = attachRoutedAbsFc(&inst->Internal.slotMoveFc);

							//Set Command Parameters
							newSlotMove->axis 					= preslot->Shuttle;
							newSlotMove->targetSlot 			= slot;

							newSlotMove->moveAbs.Axis			= &newSlotMove->axis;
							newSlotMove->moveAbs.Sector	 		= (McSectorType*)(newSlotMove->targetSlot->Sector);
							newSlotMove->moveAbs.Position	 	= newSlotMove->targetSlot->Position;
							newSlotMove->moveAbs.Velocity 		= inst->Velocity;
							newSlotMove->moveAbs.Acceleration 	= inst->Acceleration;
							newSlotMove->moveAbs.Deceleration 	= inst->Deceleration;
							newSlotMove->moveAbs.AdvancedParameters = inst->AdvancedParameters;

							newSlotMove->moveAbs.Execute 		= TRUE;

							//Clear PreslotInformation and Status
							preslot->Interface					= E_SLOT_IDLE;
							brsmemset((UDINT)&preslot->Shuttle, 0, sizeof(McAxisType));
						}
					}
					else if (preslot->Interface != E_SLOT_IDLE && preslot->Interface != E_SLOT_MANUAL)
					{
						break;
					}
				}
			}

			if (inst->CountOfShuttle == 0)
				inst->ErrorID = MyTrakIdle;
			else
				inst->ErrorID = MyTrakRun;
		}
		else
		{
			inst->ErrorID = MyTrakManual;
		}

		//Execute Slot Transfer Function
		inst->CountOfShuttle = execMyTrakSlotTrans(&inst->Internal.slotMoveFc);
	}
	else if (inst->Enable == FALSE && inst->Active == FALSE)
	{ //Disabled
		releaseMyTrakSlotTran(&inst->Internal.slotMoveFc);
		inst->ErrorID = MyTrakDisabled;
	}
}
```

#### MyTrak_Serialize.c - Move shuttles from source stage to target sector
```c
/********************************************************************
 * COPYRIGHT -- B&R Korea
 ********************************************************************
 * File: MyTrak_Serialize.c
 * Author: Taeryoung Ok
 * Created: 2021/11/06
 ********************************************************************
 * Description: Transfer Shuttles from Source Stage to Target Point of Sector
 ********************************************************************/

#include <bur/plctypes.h>
#ifdef __cplusplus
	extern "C"
	{
#endif
	#include "MyTrak.h"
	#include "MyTrakFunc.h"
#ifdef __cplusplus
	};
#endif

#define NULL 0
#define FALSE 0
#define TRUE 1

void MyTrak_Serialize(struct MyTrak_Serialize* inst)
{
	int loop = 0,prestage;

	MyTrakSlotType* slot;

	MyTrakSerializeType* newSerialMove;

	if (inst->Enable == TRUE && inst->Active == FALSE)
	{	//Disabled -> Enabled
		inst->Active = TRUE;
	}
	else if (inst->Enable == FALSE && inst->Active == TRUE)
	{	//Enabled -> Disabled
		inst->Active = FALSE;
		inst->Internal.manualCmd.CLK = FALSE; R_TRIG(&inst->Internal.manualCmd);

		releaseMyTrakSerialize(&inst->Internal.serialMoveFc);
	}
	else if (inst->Enable == TRUE && inst->Active == TRUE)
	{	//Enabled
		//Manual Command Checking
		inst->Internal.manualCmd.CLK = inst->Manual; R_TRIG(&inst->Internal.manualCmd);

		if (inst->Process == TRUE || inst->Internal.manualCmd.Q)
		{
			for (prestage = 0; prestage < 10; prestage++)
			{
				for (loop = inst->SourceSlotCount[prestage] - 1; loop >= 0; loop--)
				{
					slot = (MyTrakSlotType*)(inst->SourceStage[prestage] + sizeof(MyTrakSlotType) * loop);

					if (slot->Interface == E_SLOT_TAKEOUT_READY ||
						(slot->Interface == E_SLOT_MANUAL && slot->Shuttle.controlif != 0))
					{
						//Get New Last Slot Transfer Structure From FcBank
						newSerialMove = attachRoutedVelFc(&inst->Internal.serialMoveFc);

						//Set Command Parameters
						newSerialMove->sourceSlot				= slot;
						newSerialMove->axis 					= slot->Shuttle;

						newSerialMove->moveVel.Axis	 			= &newSerialMove->axis;
						newSerialMove->moveVel.Sector	 		= inst->TargetSector;
						newSerialMove->moveVel.Position	 		= inst->TargetPosition;
						newSerialMove->moveVel.RouteVelocity 	= inst->RoutedVelocity;
						newSerialMove->moveVel.Velocity 		= inst->Velocity;
						newSerialMove->moveVel.Acceleration 	= inst->Acceleration;
						newSerialMove->moveVel.Deceleration 	= inst->Deceleration;
						newSerialMove->moveVel.AdvancedParameters = inst->AdvancedParameters;

						newSerialMove->moveVel.Execute		 	= TRUE;

						//Clear PreslotInformation and Status
						slot->Interface							= E_SLOT_IDLE;
						brsmemset((UDINT)&slot->Shuttle, 0, sizeof(McAxisType));
					}
				}
			}

			if (inst->Internal.serialMoveFc == NULL)
				inst->ErrorID = MyTrakIdle;
			else
				inst->ErrorID = MyTrakRun;
		}
		else if (inst->Process == FALSE)
		{
			inst->ErrorID = MyTrakManual;
		}

		//Execute Serialize Function
		inst->CountOfShuttle = execMyTrakSerialize(&inst->Internal.serialMoveFc);
	}
	else if (inst->Enable == FALSE && inst->Active == FALSE)
	{	//Disabled
		releaseMyTrakSerialize(&inst->Internal.serialMoveFc);
		inst->ErrorID = MyTrakDisabled;
	}
}
```

#### MyTrak_ShInfeeder.c - Shuttle Feeding System
```c
#include <bur/plctypes.h>
#ifdef __cplusplus
	extern "C"
	{
#endif
	#include "MyTrak.h"
#ifdef __cplusplus
	};
#endif

#define NULL 0
#define FALSE 0
#define TRUE 1

void MyTrak_ShInfeeder(struct MyTrak_ShInfeeder* inst)
{
	if (inst->Enable == TRUE && inst->Active == FALSE)
	{ //Disabled -> Enable
		inst->Active = TRUE;
	}
	else if (inst->Enable == FALSE && inst->Active == TRUE)
	{ //Enabled -> Disable
		inst->Active = FALSE;
	}
	else if (inst->Enable == TRUE && inst->Active == TRUE)
	{ //Enabled
		inst->Internal.BarReadInfo.Enable = TRUE;

		if (inst->Process == TRUE)
		{
			//Auto Feeding
			if (inst->Internal.Tmr.Q == TRUE && inst->Pause == FALSE &&
				inst->Internal.BarReadInfo.BarrierInfo.RemainingTickets <= (UDINT)inst->CountOfOneShot)
			{
				inst->Internal.BarCmd.Command 	= mcACPTRAK_BARRIER_ADD_TICKETS;
				inst->Internal.BarCmd.Execute 	= TRUE;
				inst->Internal.BarCmd.AdvancedParameters.TicketCount = (DINT)inst->CountOfOneShot;

				inst->Internal.Tmr.IN 			= FALSE;
			}
			else
			{
				inst->Interval 					= 60000.0 / ((float)inst->SetPPM / (float)inst->CountOfOneShot);

				inst->Internal.Tmr.IN 			= TRUE;
				inst->Internal.Tmr.PT 			= inst->Interval;
			}
			inst->ErrorID 	= MyTrakRun;
		}
		else
		{
			//Manual Feeding
			if (inst->Internal.manualCmd.Q == TRUE)
			{
				inst->Internal.BarCmd.Command 	= mcACPTRAK_BARRIER_ADD_TICKETS;
				inst->Internal.BarCmd.Execute 	= TRUE;
				inst->Internal.BarCmd.AdvancedParameters.TicketCount = 1;

				inst->Internal.Tmr.IN 			= FALSE;
			}
			inst->Internal.Tmr.IN 			= FALSE;

			inst->ErrorID 	= MyTrakIdle;
		}
	}
	else if (inst->Enable == FALSE && inst->Active == FALSE)
	{ //Disabled
		inst->ErrorID 	= MyTrakDisabled;
	}

	inst->Internal.manualCmd.CLK = inst->Manual;
	R_TRIG(&inst->Internal.manualCmd);

	if (inst->Internal.BarCmd.Done == TRUE)
		inst->Internal.BarCmd.Execute = FALSE;

	inst->Internal.BarCmd.ProcessPoint		= inst->ProcessPoint;
	inst->Internal.BarReadInfo.ProcessPoint	= inst->ProcessPoint;

	TON(&inst->Internal.Tmr);
	MC_BR_BarrierCommand_AcpTrak(&inst->Internal.BarCmd);
	MC_BR_BarrierReadInfo_AcpTrak(&inst->Internal.BarReadInfo);
}
```

#### MyTrak_TicketArea.c - Keep shuttles count between two process point
```c
#include <bur/plctypes.h>
#ifdef __cplusplus
	extern "C"
	{
#endif
	#include "MyTrak.h"
#ifdef __cplusplus
	};
#endif

#define FALSE 0
#define TRUE 1

void MyTrak_TicketArea(struct MyTrak_TicketArea* inst)
{
	if (inst->Enable == TRUE && inst->Active == FALSE)
	{
		inst->Internal.fbInEnable.Enable 			= TRUE;
		inst->Internal.fbOutEnable.Enable 			= TRUE;
		inst->Internal.fbBarrierReadInfo.Enable 	= TRUE;

		if (inst->Internal.fbInEnable.Valid == TRUE && inst->Internal.fbOutEnable.Valid == TRUE &&
			inst->Internal.fbOutEnable.Valid == TRUE)
		{
			inst->Internal.fbBarrier.Execute		= TRUE;
			inst->Internal.fbBarrier.Command 		= mcACPTRAK_BARRIER_ADD_TICKETS;
			inst->Internal.fbBarrier.AdvancedParameters.TicketCount = inst->MaximumShuttleCount;

			if (inst->Internal.fbBarrier.Done == TRUE)
			{
				inst->Internal.fbBarrier.Execute	= FALSE;
				inst->Active 						= TRUE;
			}
		}
	}
	else if (inst->Enable == TRUE && inst->Active == TRUE)
	{
		if (inst->Internal.fbOutGetInfo.Done == FALSE)
		{
			if (inst->Internal.fbOutEnable.EventCount > 0)
				inst->Internal.fbOutGetInfo.Execute = TRUE;
		}
		else if (inst->Internal.fbInGetInfo.Done == FALSE)
		{
			if (inst->Internal.fbInEnable.EventCount > 0)
				inst->Internal.fbInGetInfo.Execute = TRUE;
//			else
//				inst->Internal.fbOutGetInfo.Execute = FALSE;
		}
		else
		{
			if (inst->Internal.fbOutGetInfo.TrgPointInfo.Axis.controlif == inst->Internal.fbInGetInfo.TrgPointInfo.Axis.controlif
				&& inst->Internal.fbOutGetInfo.TrgPointInfo.Axis.controlif != 0
				&&inst->Internal.fbInGetInfo.TrgPointInfo.Axis.controlif != 0)
			{
//				if (inst->Internal.fbBarrierReadInfo.BarrierInfo.RemainingTickets + inst->Internal.fbInEnable.EventCount
//					< inst->MaximumShuttleCount)
//				{
					inst->Internal.fbBarrier.Execute		= TRUE;
					inst->Internal.fbBarrier.Command 		= mcACPTRAK_BARRIER_ADD_TICKETS;
					inst->Internal.fbBarrier.AdvancedParameters.TicketCount = 1;
//				}

				if (inst->Internal.fbBarrier.Done == TRUE)
				{
					inst->Internal.fbBarrier.Execute		= FALSE;
					inst->Internal.fbInGetInfo.Execute 		= FALSE;
					inst->Internal.fbOutGetInfo.Execute 	= FALSE;
				}
			}
			else
			{
				inst->Internal.fbOutGetInfo.Execute = FALSE;
			}
		}
	}
	else if (inst->Enable == FALSE && inst->Active == TRUE)
	{
		inst->Active 								= FALSE;
	}
	else if (inst->Enable == FALSE && inst->Active == FALSE)
	{
		inst->Internal.fbInEnable.Enable 			= FALSE;
		inst->Internal.fbOutEnable.Enable 			= FALSE;
		inst->Internal.fbBarrierReadInfo.Enable 	= TRUE;

		if (inst->Internal.fbBarrier.Done == TRUE)
		{
			inst->Internal.fbBarrier.Execute 	= FALSE;
		}
		else if (inst->Internal.fbBarrierReadInfo.BarrierInfo.Status != mcACPTRAK_BARRIER_OPENED)
		{
			inst->Internal.fbBarrier.Command 	= mcACPTRAK_BARRIER_OPEN;
			inst->Internal.fbBarrier.Execute 	= TRUE;
		}
	}

	inst->Internal.fbInEnable.ProcessPoint 		 	= inst->InPoint;
	inst->Internal.fbInGetInfo.ProcessPoint 		= inst->InPoint;

	MC_BR_TrgPointEnable_AcpTrak(&inst->Internal.fbInEnable);
	MC_BR_TrgPointGetInfo_AcpTrak(&inst->Internal.fbInGetInfo);

	inst->Internal.fbOutEnable.ProcessPoint			= inst->OutPoint;
	inst->Internal.fbOutGetInfo.ProcessPoint		= inst->OutPoint;

	MC_BR_TrgPointEnable_AcpTrak(&inst->Internal.fbOutEnable);
	MC_BR_TrgPointGetInfo_AcpTrak(&inst->Internal.fbOutGetInfo);

	inst->Internal.fbBarrier.ProcessPoint 			= inst->InPoint;
	inst->Internal.fbBarrierReadInfo.ProcessPoint 	= inst->InPoint;
	MC_BR_BarrierReadInfo_AcpTrak(&inst->Internal.fbBarrierReadInfo);
	MC_BR_BarrierCommand_AcpTrak(&inst->Internal.fbBarrier);
}
```

#### MyTrak_ChangeVel.c - ChangeVelcity in specific process point
```c
#include <bur/plctypes.h>
#ifdef __cplusplus
	extern "C"
	{
#endif
	#include "MyTrak.h"
#ifdef __cplusplus
	};
#endif

#define TRUE 1
#define FALSE 0

/* TODO: Add your comment here */
void MyTrak_ChangeVel(struct MyTrak_ChangeVel* inst)
{
	switch(inst->Internal.step)
	{
		case 0:
			if (inst->Enable == TRUE)
			{
				inst->Internal.TrgEnable.Enable = TRUE;

				if (inst->Internal.TrgEnable.Valid)
					inst->Internal.step = 100;
			}
			break;

		case 100:
			if (inst->Internal.TrgEnable.EventCount > 0)
			{
				inst->Internal.TrgGetInfo.Execute = TRUE;
				inst->Internal.step = 200;
			}
			break;

		case 200:
			if (inst->Internal.TrgGetInfo.Done == TRUE)
			{
				inst->Internal.ElasticMoveVel.Axis 			= (McAxisType*)&inst->Internal.TrgGetInfo.TrgPointInfo.Axis;

				inst->Internal.ElasticMoveVel.Velocity 		= inst->Velocity;
				inst->Internal.ElasticMoveVel.Acceleration 	= inst->Acceleration;
				inst->Internal.ElasticMoveVel.Deceleration 	= inst->Deceleration;
				inst->Internal.ElasticMoveVel.Direction 	= inst->Direction;
				inst->Internal.ElasticMoveVel.Execute	 	= TRUE;

				if ((inst->Internal.ElasticMoveVel.Active == TRUE && inst->Internal.preActive == FALSE)
				|| inst->Internal.ElasticMoveVel.Error == TRUE)
				{
					inst->Internal.TrgGetInfo.Execute 		= FALSE;
					inst->Internal.ElasticMoveVel.Execute	= FALSE;
					inst->Internal.step 					= 100;
				}
			}
			break;
	}

	inst->Internal.TrgEnable.ProcessPoint = inst->ProcessPoint;
	inst->Internal.TrgGetInfo.ProcessPoint = inst->ProcessPoint;
	inst->Internal.preActive = inst->Internal.ElasticMoveVel.Active;

	MC_BR_TrgPointEnable_AcpTrak(&inst->Internal.TrgEnable);
	MC_BR_TrgPointGetInfo_AcpTrak(&inst->Internal.TrgGetInfo);
	MC_BR_ElasticMoveVel_AcpTrak(&inst->Internal.ElasticMoveVel);
}
```

#### MyTrak_UntilStop.c - Not Implemented
```c
#include <bur/plctypes.h>
#ifdef __cplusplus
	extern "C"
	{
#endif
	#include "MyTrak.h"
	#include "MyTrakFunc.h"
#ifdef __cplusplus
	};
#endif

#define NULL 0
#define FALSE 0
#define TRUE 1

void MyTrak_UntilStop(struct MyTrak_UntilStop* inst)
{
	MyTrakSerializeType* newSerialMove;

	if (inst->Execute == TRUE && inst->Active == FALSE)
	{
		inst->Internal.getShuttle.Sector 							= inst->SourceSector;

		inst->Internal.getShuttle.AdvancedParameters.StartPosition 	= inst->SourceStart;
		inst->Internal.getShuttle.AdvancedParameters.EndPosition 	= inst->SourceEnd;

		inst->Internal.getShuttle.Enable = TRUE;

		inst->Active = TRUE;
	}
	else if (inst->Execute == FALSE && inst->Active == TRUE)
	{
	}
	else if (inst->Execute == TRUE && inst->Active == TRUE)
	{
		if (inst->Internal.getShuttle.Valid == TRUE && inst->Internal.getShuttle.RemainingCount > 0)
		{
			if (inst->Internal.getShuttle.RemainingCount + inst->CountOfShuttle < inst->Internal.getShuttle.TotalCount)
			{
				newSerialMove = attachRoutedVelFc(&inst->Internal.serialMoveFc);
				newSerialMove->axis = inst->Internal.getShuttle.Axis;

				newSerialMove->moveVel.Axis 				= &newSerialMove->axis;

				newSerialMove->moveVel.Sector 				= inst->TargetSector;
				newSerialMove->moveVel.Position 			= inst->TargetPosition;
				newSerialMove->moveVel.RouteVelocity 		= inst->RoutedVelocity;
				newSerialMove->moveVel.Velocity 			= inst->Velocity;
				newSerialMove->moveVel.Acceleration 		= inst->Acceleration;
				newSerialMove->moveVel.Deceleration 		= inst->Deceleration;
				newSerialMove->moveVel.AdvancedParameters 	= inst->AdvancedParameters;

				newSerialMove->moveVel.Execute 				= TRUE;

				inst->Internal.getShuttle.Next = FALSE;

				inst->CountOfShuttle++;
			}
			else
			{
				inst->Internal.getShuttle.Next = TRUE;
			}
		}
		else
		{

		}
		execMyTrakSerialize(&inst->Internal.serialMoveFc);
	}
}
```

#### CheckProcessStatus.c - Check all slot's status
```c
#include <bur/plctypes.h>
#ifdef __cplusplus
	extern "C"
	{
#endif
	#include "MyTrak.h"
#ifdef __cplusplus
	};
#endif

#define FALSE 0
#define TRUE 1

plcbit GetTakeOutReady(unsigned long Stage, unsigned char CountofSlots)
{
	int 				loop;
	MyTrakSlotType* 	slot;

	for (loop = 0; loop < CountofSlots; loop++)
	{
		slot = (MyTrakSlotType*)(Stage + sizeof(MyTrakSlotType) * loop);

		if (slot->Interface != E_SLOT_MANUAL && slot->Interface != E_SLOT_TAKEOUT_READY)
			return FALSE;
	}
	return TRUE;
}

plcbit GetProcessReady(unsigned long Stage, unsigned char CountofSlots)
{
	int 				loop;
	MyTrakSlotType* 	slot;

	for (loop = 0; loop < CountofSlots; loop++)
	{
		slot = (MyTrakSlotType*)(Stage + sizeof(MyTrakSlotType) * loop);

		if (slot->Interface != E_SLOT_MANUAL && slot->Interface != E_SLOT_PROCESS_READY)
			return FALSE;
	}
	return TRUE;
}

plcbit GetProcessing(unsigned long Stage, unsigned char CountofSlots)
{
	int 				loop;
	MyTrakSlotType* 	slot;

	for (loop = 0; loop < CountofSlots; loop++)
	{
		slot = (MyTrakSlotType*)(Stage + sizeof(MyTrakSlotType) * loop);

		if (slot->Interface != E_SLOT_MANUAL && slot->Interface != E_SLOT_PROCESSING)
			return FALSE;
	}
	return TRUE;
}

E_SLOT_IF_STATE GetStageStatus(unsigned long Stage, unsigned char CountofSlots)
{
	int 				loop;
	MyTrakSlotType* 	slot;
	MyTrakSlotType* 	preslot;

	for (loop = 1; loop < CountofSlots; loop++)
	{
		slot = (MyTrakSlotType*)(Stage + sizeof(MyTrakSlotType) * loop);
		preslot = (MyTrakSlotType*)(Stage + sizeof(MyTrakSlotType) * (loop - 1));

		if (slot->Interface != preslot->Interface)
			return E_SLOT_UNKNOWN;
	}
	return preslot->Interface;
}
```

#### InitializeFunctionblockBank.c - Initializa & Get/Return AbsMove FunctionBlock
```c
/********************************************************************
 * COPYRIGHT -- B&R Korea
 ********************************************************************
 * File: InitializeFunctionblockBank.c
 * Author: Taeryoung Ok
 * Created: 2021/11/07
 ********************************************************************
 * Description: Functions for Functionblock Banking System
 ********************************************************************/

#include <bur/plctypes.h>
#ifdef __cplusplus
	extern "C"
	{
#endif
#include "MyTrak.h"
#include "AsBrStr.h"
#include "sys_lib.h"
#include "MyTrakFunc.h"
#ifdef __cplusplus
	};
#endif

#define NULL 0
#define FALSE 0
#define TRUE 1

MyTrakSlotTransType defaultSlotTransFc;
MyTrakSerializeType defaultSerializeFc;

UDINT _adrRoutedAbsFunc = 0;
UDINT _adrRoutedVelFunc = 0;

plcbit InitializeFcBank(unsigned short shuttleCount)
{
	int loop = 0;
	MyTrakSlotTransType* routedAbsFc;
	MyTrakSerializeType* routedVelFc;

	if (shuttleCount == 0)
	{
		return FALSE;
	}
	else
	{
		TMP_alloc((UDINT)sizeof(MyTrakSlotTransType), (void*)&_adrRoutedAbsFunc);
		brsmemcpy((UDINT)_adrRoutedAbsFunc, (UDINT)&defaultSlotTransFc, (UDINT)sizeof(MyTrakSlotTransType));

		TMP_alloc((UDINT)sizeof(MyTrakSerializeType), (void*)&_adrRoutedVelFunc);
		brsmemcpy((UDINT)_adrRoutedVelFunc, (UDINT)&defaultSerializeFc, (UDINT)sizeof(MyTrakSerializeType));
	}

	routedAbsFc = (MyTrakSlotTransType*)_adrRoutedAbsFunc;

	for (loop = 1; loop < shuttleCount; loop++)
	{
		TMP_alloc(sizeof(MyTrakSlotTransType), (void*)&routedAbsFc->next);
		brsmemcpy((UDINT)routedAbsFc->next, (UDINT)&defaultSlotTransFc, (UDINT)sizeof(MyTrakSlotTransType));
		routedAbsFc = routedAbsFc->next;
	}

	routedVelFc = (MyTrakSerializeType*)_adrRoutedVelFunc;

	for (loop = 1; loop < shuttleCount; loop++)
	{
		TMP_alloc(sizeof(MyTrakSerializeType), (void*)&routedVelFc->next);
		brsmemcpy((UDINT)routedVelFc->next, (UDINT)&defaultSerializeFc, (UDINT)sizeof(MyTrakSerializeType));
		routedVelFc = routedVelFc->next;
	}
	return TRUE;
}

MyTrakSlotTransType* rentRoutedAbsFc()
{
	MyTrakSlotTransType* returnValue;

	returnValue 		= (MyTrakSlotTransType*)_adrRoutedAbsFunc;
	_adrRoutedAbsFunc 	= (UDINT)((MyTrakSlotTransType*)_adrRoutedAbsFunc)->next;
	returnValue->next 	= 0;

	return returnValue;
}

MyTrakSlotTransType* attachRoutedAbsFc(MyTrakSlotTransType** rootSlotMove)
{
	MyTrakSlotTransType* returnValue = *rootSlotMove;

	if (returnValue == NULL)
	{
		(*rootSlotMove) = rentRoutedAbsFc();
		return (*rootSlotMove);
	}
	else
	{
		while (returnValue->next != NULL)
			returnValue = returnValue->next;

		returnValue->next = rentRoutedAbsFc();

		return returnValue->next;
	}
}

void rtnRoutedAbsFc(MyTrakSlotTransType* rtnFc)
{
	rtnFc->moveAbs.Axis 		= NULL;
	rtnFc->moveAbs.Sector 		= NULL;
	rtnFc->moveAbs.Execute 		= FALSE;

	MC_BR_RoutedMoveAbs_AcpTrak(&rtnFc->moveAbs);
	rtnFc->next 		= (MyTrakSlotTransType*)_adrRoutedAbsFunc;
	_adrRoutedAbsFunc 	= (UDINT)rtnFc;
}

MyTrakSerializeType* rentRoutedVelFc()
{
	MyTrakSerializeType* returnValue;

	returnValue 		= (MyTrakSerializeType*)_adrRoutedVelFunc;
	_adrRoutedVelFunc 	= (UDINT)((MyTrakSerializeType*)_adrRoutedVelFunc)->next;
	returnValue->next 	= 0;

	return returnValue;
}

MyTrakSerializeType* attachRoutedVelFc(MyTrakSerializeType** rootSerialize)
{
	MyTrakSerializeType* returnValue = *rootSerialize;

	if (returnValue == NULL)
	{
		(*rootSerialize) = rentRoutedVelFc();
		return (*rootSerialize);
	}
	else
	{
		while (returnValue->next != NULL)
			returnValue = returnValue->next;

		returnValue->next = rentRoutedVelFc();

		return returnValue->next;
	}
}

void rtnRoutedVelFc(MyTrakSerializeType* rtnFc)
{
	rtnFc->moveVel.Axis 		= NULL;
	rtnFc->moveVel.Sector 		= NULL;
	rtnFc->moveVel.Execute 		= FALSE;

	MC_BR_RoutedMoveVel_AcpTrak(&rtnFc->moveVel);
	rtnFc->next 		= (MyTrakSerializeType*)_adrRoutedVelFunc;
	_adrRoutedVelFunc 	= (UDINT)rtnFc;
}

int SearchNextSlot(UDINT firstSlot, int currentSlot, unsigned int slotCount)
{
	int loop = 0;

	MyTrakSlotType* slot = 0;

	for (loop = currentSlot - 1; loop >= 0; loop--)
	{
		slot = (MyTrakSlotType*)(firstSlot + sizeof(MyTrakSlotType) * loop);

		if (slot->Enable == TRUE)
			return loop;
	}

	for (loop = slotCount - 1; loop >= currentSlot; loop--)
	{
		slot = (MyTrakSlotType*)(firstSlot + sizeof(MyTrakSlotType) * loop);

		if (slot->Enable == TRUE)
			return loop;
	}
	return -1;
}

DINT execMyTrakSlotTrans(MyTrakSlotTransType** executeList)
{
	DINT returnValue = 0;

	if (*executeList == NULL) return 0;

	//Execute Slot Transfer Function
	MyTrakSlotTransType* preSlotMove 	= NULL;
	MyTrakSlotTransType* slotMove 		= *executeList;

	while (slotMove != 0)
	{
		//Execution
		MC_BR_RoutedMoveAbs_AcpTrak(&slotMove->moveAbs);

		if (slotMove->moveAbs.Done == TRUE)
		{ //Move Done Case
			//Slot Information
			slotMove->targetSlot->Shuttle 		= slotMove->axis;

			if (slotMove->targetSlot->Interface == E_SLOT_IDLE)
				slotMove->targetSlot->Interface 	= E_SLOT_PROCESS_READY;

			//Reconection List and Return to bank
			if (preSlotMove != NULL)
			{
				preSlotMove->next 	= slotMove->next;
				rtnRoutedAbsFc(slotMove);
				slotMove			= preSlotMove->next;
			}
			else if (preSlotMove == NULL && slotMove->next != NULL)
			{
				(*executeList) 		= slotMove->next;
				rtnRoutedAbsFc(slotMove);
				slotMove			= (*executeList);
			}
			else if (preSlotMove == NULL && slotMove->next == NULL)
			{
				(*executeList) 		= NULL;
				rtnRoutedAbsFc(slotMove);
				slotMove			= NULL;
			}
		}
		else if (slotMove->moveAbs.CommandAborted == TRUE)
		{ //Move Abort Case
			slotMove->moveAbs.Execute 			= FALSE;
		}
		else if (slotMove->moveAbs.Error == TRUE)
		{ //Move Error Case

		}
		else
		{
			preSlotMove = slotMove;
			slotMove 	= slotMove->next;
		}
		returnValue++;
	}
	return returnValue;
}

void releaseMyTrakSlotTran(MyTrakSlotTransType** executeList)
{
	if (*executeList == NULL) return;

	//Execute Slot Transfer Function
	MyTrakSlotTransType* tmpSlotMove 	= NULL;
	MyTrakSlotTransType* slotMove 		= *executeList;

	while (slotMove != 0)
	{
		//Return FunctionBlock
		tmpSlotMove 		= slotMove->next;
		rtnRoutedAbsFc(slotMove);
		slotMove 			= tmpSlotMove;
	}
	*executeList = NULL;

	return;
}

DINT execMyTrakSerialize(MyTrakSerializeType** executeList)
{
	DINT returnValue = 0;

	if (*executeList == NULL) return 0;

	MyTrakSerializeType* preSerialMove 	= NULL;
	MyTrakSerializeType* serialMove		= *executeList;

	while (serialMove != 0)
	{
		//Execution
		MC_BR_RoutedMoveVel_AcpTrak(&serialMove->moveVel);

		//Execution Check
		if (serialMove->moveVel.PositionReached == TRUE ||
			serialMove->moveVel.CommandAborted == TRUE)
		{
			//Reconection List and Return to bank
			if (preSerialMove != NULL)
			{
				preSerialMove->next = serialMove->next;
				rtnRoutedVelFc(serialMove);
				serialMove = preSerialMove->next;
			}
			else if (preSerialMove == NULL && serialMove->next != NULL)
			{
				(*executeList) = serialMove->next;
				rtnRoutedVelFc(serialMove);
				serialMove = (*executeList);
			}
			else if (preSerialMove == NULL && serialMove->next == NULL)
			{
				(*executeList) = NULL;
				rtnRoutedVelFc(serialMove);
				serialMove = NULL;
			}
		}
		else
		{
			preSerialMove 	= serialMove;
			serialMove 		= serialMove->next;
		}
		returnValue++;
	}
	return returnValue;
}

void releaseMyTrakSerialize(MyTrakSerializeType** executeList)
{
	if (*executeList == NULL) return;

	//Execute Slot Transfer Function
	MyTrakSerializeType* tmpSlotMove 	= NULL;
	MyTrakSerializeType* slotMove		= *executeList;

	while (slotMove != 0)
	{
		//Return FunctionBlock
		tmpSlotMove 		= slotMove->next;
		rtnRoutedVelFc(slotMove);
		slotMove 			= tmpSlotMove;
	}

	*executeList = NULL;

	return;
}
```

#### Random.c
```c
#include <bur/plctypes.h>
#ifdef __cplusplus
	extern "C"
	{
#endif
	#include "MyTrak.h"
	#include "stdlib.h"
#ifdef __cplusplus
	};
#endif

#define FALSE 0
#define TRUE 1

plcbit Random(float Percent)
{
 	unsigned int test = rand();
	double result;

	result = (double)test/(double)4294967295.0 * (double)100.0;

	return result < (double)Percent ? TRUE : FALSE;
}
```

### Library Logical/Libraries/MyTime (ANSIC)
Depends on: AsBrStr, sys_lib

#### Types.typ - Exported data types
```iecst
TYPE
	MyTime_TimeCheck_Internal_type : 	STRUCT
		rtcTime : RTCtime_typ;
		last_cycle_start : RTCtime_typ;
		maxCycle : RTCtime_typ;
		lastCycle : RTCtime_typ;
	END_STRUCT;
END_TYPE
```

#### MyTime.fun - Exported functions and function blocks
```iecst
{REDUND_ERROR} FUNCTION_BLOCK MyTime_TimeCheck (*TODO: Add your comment here*)
	VAR_OUTPUT
		Time : REAL;
	END_VAR
	VAR
		Internal : MyTime_TimeCheck_Internal_type;
	END_VAR
END_FUNCTION_BLOCK
```

#### MyTime_TimeCheck.c
```c
#include <bur/plctypes.h>
#ifdef __cplusplus
	extern "C"
	{
#endif
	#include "MyTime.h"
#ifdef __cplusplus
	};
#endif

#define FALSE 0
#define TRUE 1

void MyTime_TimeCheck(struct MyTime_TimeCheck* inst)
{
	/* Get time */
	RTC_gettime(&inst->Internal.rtcTime);

	/* Calculate the cycle time */
	if(inst->Internal.rtcTime.year == 0)
	{
		/* Store the last time */
		inst->Internal.last_cycle_start = inst->Internal.rtcTime;
	}else{
		/* Clear the last cycle information */
		brsmemset(&inst->Internal.lastCycle,0,sizeof(inst->Internal.lastCycle));
		/* Create local counting variables */
		unsigned int SecCnt = 0;
		unsigned int MinCnt = 0;
		unsigned int HrCnt = 0;
		unsigned int DayCnt = 0;
		unsigned int MonCnt = 0;
		unsigned int YrCnt = 0;

		/* Start with microseconds */
		inst->Internal.lastCycle.microsec = inst->Internal.rtcTime.microsec;
		/* Miliseconds calculation */
		if(inst->Internal.rtcTime.millisec < inst->Internal.last_cycle_start.millisec){
			inst->Internal.lastCycle.millisec = ((inst->Internal.rtcTime.millisec+1000)-inst->Internal.last_cycle_start.millisec);
			SecCnt = 1;
		}else{
			inst->Internal.lastCycle.millisec = (inst->Internal.rtcTime.millisec-inst->Internal.last_cycle_start.millisec);
		}
		// Second calculation
		if(inst->Internal.rtcTime.second < inst->Internal.last_cycle_start.second){
			inst->Internal.lastCycle.second = ((inst->Internal.rtcTime.second+60)-inst->Internal.last_cycle_start.second)-SecCnt;
			MinCnt = 1;
		}else{
			inst->Internal.lastCycle.second = (inst->Internal.rtcTime.second-inst->Internal.last_cycle_start.second)-SecCnt;
		}
		// Minute calculation
		if(inst->Internal.rtcTime.minute < inst->Internal.last_cycle_start.minute){
			inst->Internal.lastCycle.minute = ((inst->Internal.rtcTime.minute+60)-inst->Internal.last_cycle_start.minute)-MinCnt;
			HrCnt = 1;
		}else{
			inst->Internal.lastCycle.minute = (inst->Internal.rtcTime.minute-inst->Internal.last_cycle_start.minute)-MinCnt;
		}
		// Hour calculation
		if(inst->Internal.rtcTime.hour < inst->Internal.last_cycle_start.hour){
			inst->Internal.lastCycle.hour = ((inst->Internal.rtcTime.hour+24)-inst->Internal.last_cycle_start.hour)-HrCnt;
			DayCnt = 1;
		}else{
			inst->Internal.lastCycle.hour = (inst->Internal.rtcTime.hour-inst->Internal.last_cycle_start.hour) -HrCnt;
		}
		// Day calculation
		if(inst->Internal.rtcTime.day < inst->Internal.last_cycle_start.day){
			inst->Internal.lastCycle.day = ((inst->Internal.rtcTime.day+30)-inst->Internal.last_cycle_start.day)-DayCnt;
			MonCnt = 1;
		}else{
			inst->Internal.lastCycle.day = (inst->Internal.rtcTime.day-inst->Internal.last_cycle_start.day)-DayCnt;
		}
		// Month calculation
		if(inst->Internal.rtcTime.month < inst->Internal.last_cycle_start.month){
			inst->Internal.lastCycle.month = ((inst->Internal.rtcTime.month+12)-inst->Internal.last_cycle_start.month)-MonCnt;
			YrCnt = 1;
		}else{
			inst->Internal.lastCycle.month = (inst->Internal.rtcTime.month-inst->Internal.last_cycle_start.month)-MonCnt;
		}
		// Year calculation
		if(inst->Internal.rtcTime.year < inst->Internal.last_cycle_start.year){
			inst->Internal.lastCycle.year = ((inst->Internal.rtcTime.year)-inst->Internal.last_cycle_start.year)-YrCnt;
		}else{
			inst->Internal.lastCycle.year = (inst->Internal.rtcTime.year-inst->Internal.last_cycle_start.year)-YrCnt;
		}

		if(inst->Internal.maxCycle.year < inst->Internal.lastCycle.year &&
			inst->Internal.maxCycle.month < inst->Internal.lastCycle.month &&
			inst->Internal.maxCycle.day < inst->Internal.lastCycle.day &&
			inst->Internal.maxCycle.hour < inst->Internal.lastCycle.hour &&
			inst->Internal.maxCycle.minute  < inst->Internal.lastCycle.minute &&
			inst->Internal.maxCycle.second < inst->Internal.lastCycle.second &&
		inst->Internal.maxCycle.millisec < inst->Internal.lastCycle.millisec){

			inst->Internal.maxCycle = inst->Internal.lastCycle;
		}

		if(inst->Internal.lastCycle.minute == 0){
			if(inst->Internal.lastCycle.second == 0){
				inst->Time = 0.001 * inst->Internal.lastCycle.millisec;

				//	Internal.tmpString := UINT_TO_STRING(Internal.lastCycle.millisec);
				//	brsstrcat(ADR(Internal.tmpString), ADR('ms'));
			}else{

				//Internal.tmpString := USINT_TO_STRING(Internal.lastCycle.second);
				//brsstrcat(ADR(Internal.tmpString), ADR('s '));
				//Internal.timeTemp := UINT_TO_STRING(Internal.lastCycle.millisec);
				//	brsstrcat(ADR(Internal.tmpString), ADR(Internal.timeTemp));
				//brsstrcat(ADR(Internal.tmpString), ADR('ms'));
				inst->Time = 0.001 * inst->Internal.lastCycle.millisec;
				inst->Time = inst->Time + 1 * inst->Internal.lastCycle.second;
			}
		}
		inst->Internal.last_cycle_start = inst->Internal.rtcTime;

	}
}
```

### gTrakSupport.var - Global variables
```iecst
(*constants*)
VAR CONSTANT
	TRAK_MAX_SHUTTLE : UINT := 100; (*maximum number of shuttles handled in this application - should be set equal or higher than Shuttles-maximum-count setting in mappMotion assembly config file*)
	TRAK_MAX_SEGMENT : UINT := 26; (*maximum number of segments handled in this application*)
	TRAK_MAX_POWER_CABLE : UINT := 7; (*maximum number of power cables handled in this application*)
	TRAK_MAX_POWER_SUPPLY : UINT := 7; (*maximum number of power supplys handled in this application*)
END_VAR
(*interface TrakDesign shuttle online interaction*)
VAR
	gTrakDesignShuttleOnline : TrakDesignShuttleOnlineType := (0);
END_VAR
(*interface TrakDesign shuttle online interaction*)
VAR CONSTANT
	COUNT_OF_SIM_SHUTTLE : USINT := 19;
	GAP_BETWEEN_OF_SHUTTLE : LREAL := 0.14;
END_VAR
```

### gTrakSupport.typ - Global data types
```iecst
(*interface TrakDesign shuttle online interaction*)

TYPE
	TrakDesignShuttleOnlineType : 	STRUCT
		CmdSetPayloadIx : BOOL; (*command to set a payload index for a shuttle*)
		CmdAddShuttle : BOOL; (*command indicating that a shuttle has been added to the trak*)
		CmdDeleteShuttle : BOOL; (*command indicating that a shuttle has been deleted from the trak*)
		CmdRecordToolData : BOOL; (*command activate recording of TrakDesign-Tool data*)
		ParaPayloadIx : USINT; (*parameter to select a payload with this index for a shuttle*)
		ParaShuttleID : UINT; (*parameter for identification of a shuttle using its ID
can be used for CmdSetPayloadIx and CmdDeleteShuttle*)
		ParaShuttleAxis : McAxisType; (*parameter for identification of a shuttle using its Axis (McAxisType)
can be used for CmdSetPayloadIx and CmdDeleteShuttle
mandatory for CmdAddShuttle*)
		Done : BOOL; (*status command done
flag is set for one cycle only*)
		TimeRecordToolDataActive : REAL; (*monitor time recording of TrakDesign-Tool data active*)
	END_STRUCT;
END_TYPE

(*internal: process-ParID read/write*)

TYPE
	TrakSegParIDProcessDataType : 	STRUCT
		Num : USINT; (*number of ParID's in this list to read/write at once*)
		Fub : ARRAY[0..19]OF McAcpTrakSegProcessParIDType; (*ParID list for FUB MC_BR_SegProcessParID_AcpTrak*)
		VarREAL : ARRAY[0..19]OF REAL; (*temporary REAL variable*)
		VarDINT : ARRAY[0..19]OF DINT; (*temporary DINT variable*)
	END_STRUCT;
END_TYPE
```

### Program Logical/Source/Utility/Vis (IEC)

#### Types.typ
```iecst
TYPE
	VisuPage_typ : 	STRUCT  (*Structure type for page control*)
		CurrenPage : UINT; (*Current page index*)
		NewPage : UINT; (*New page index*)
		SetOldPage : UINT; (*Set old page page index*)
		SetPage : UINT; (*Set page index*)
		StartingBar : UINT; (*Starting page bar graph*)
		TON_Boot : TON; (*Timer for bar graph in booting page *)
		BootingText : USINT; (*Text for description in booting page*)
	END_STRUCT;
END_TYPE
```

#### Variables.var
```iecst
VAR
	Vis : McAcpTrakAssemblyVisData;
	SizeofVis : UDINT := 0;
	NumVisShuttle : USINT := 0;
	i : USINT := 0;
	pUserData : REFERENCE TO ShuttleUserData_typ;
	PageCon : VisuPage_typ;
END_VAR
```

#### Main.st
```iecst
PROGRAM _INIT

    // size of Vis structure - this value has to be entered in B&R scene viewer (PVI -> Options -> Size)
	SizeofVis := SIZEOF(Vis);
	// max number of displayed shuttles
	NumVisShuttle := SIZEOF(Vis.Shuttle) / SIZEOF(Vis.Shuttle[0]);

END_PROGRAM

PROGRAM _CYCLIC

	FOR i:=0 TO (NumVisShuttle-1) DO
		IF gShuttleMon.Shuttle[i].Available THEN
			// format selected monitor data to fit B&R scene viewer
			Vis.Shuttle[i].Available     := 1;
			Vis.Shuttle[i].PositionX     := LREAL_TO_REAL(gShuttleMon.Shuttle[i].Position.X);
			Vis.Shuttle[i].PositionY     := LREAL_TO_REAL(gShuttleMon.Shuttle[i].Position.Y);
			Vis.Shuttle[i].RotationZ     := LREAL_TO_REAL(gShuttleMon.Shuttle[i].Orientation.Angle1);
			Vis.Shuttle[i].ExtentToFront := LREAL_TO_REAL(gShuttleMon.Shuttle[i].ExtentToFront);
			Vis.Shuttle[i].ExtentToBack  := LREAL_TO_REAL(gShuttleMon.Shuttle[i].ExtentToBack);
			Vis.Shuttle[i].Width         := LREAL_TO_REAL(gShuttleMon.Shuttle[i].Width);
			brsitoa(gShuttleMon.Shuttle[i].Index, ADR(Vis.Shuttle[i].Text));
			Vis.Shuttle[i].ColorRed      := 0.5;       //
			Vis.Shuttle[i].ColorGreen    := 0.5;      // default shuttle color gray
			Vis.Shuttle[i].ColorBlue     := 0.5;        //

			// example: set shuttle colour via user data
			IF gShuttleMon.Shuttle[i].UserData <> 0 THEN
				pUserData ACCESS gShuttleMon.Shuttle[i].UserData;    // access to user data of this shuttle
			(*	IF pUserData.Color = ORANGE THEN                     // Color is defined with RGB values between 0 and 1
					Vis.Shuttle[i].ColorRed     := 1.000;
					Vis.Shuttle[i].ColorGreen   := 0.5451;
					Vis.Shuttle[i].ColorBlue    := 0.000;
				ELSIF pUserData.Color = GREEN THEN
					Vis.Shuttle[i].ColorRed     := 0.000;
					Vis.Shuttle[i].ColorGreen   := 1.000;
					Vis.Shuttle[i].ColorBlue    := 0.000;
				ELSIF pUserData.Color = RED THEN
					Vis.Shuttle[i].ColorRed     := 1.000;
					Vis.Shuttle[i].ColorGreen   := 0.000;
					Vis.Shuttle[i].ColorBlue    := 0.000;
				ELSIF pUserData.Color = BLUE THEN
					Vis.Shuttle[i].ColorRed     := 0.000;
					Vis.Shuttle[i].ColorGreen   := 0.000;
					Vis.Shuttle[i].ColorBlue    := 1.000;
				ELSIF pUserData.Color = WHITE THEN
					Vis.Shuttle[i].ColorRed     := 1.000;
					Vis.Shuttle[i].ColorGreen   := 1.000;
					Vis.Shuttle[i].ColorBlue    := 1.000;
				END_IF  *)
			END_IF

		ELSE
			brsmemset(ADR(Vis.Shuttle[i]), 0, SIZEOF(Vis.Shuttle[0]));  //If the selected shuttle is not available, it will be invisible in the Scene Viewer
		END_IF
	END_FOR

	// Page control
	IF PageCon.NewPage = 65535 AND PageCon.SetPage <> PageCon.SetOldPage THEN
		IF PageCon.SetPage = 0 THEN
			PageCon.SetPage		:= PageCon.SetOldPage;
		ELSE
			PageCon.NewPage		:= PageCon.SetPage;
			PageCon.SetOldPage	:= PageCon.SetPage;
		END_IF
	END_IF

END_PROGRAM
```

### Program Logical/Source/Utility/Simulation (IEC) - Shuttle Attach

#### Variables.var
```iecst
(**)
VAR CONSTANT
	SIM_POWER_ON : INT := 0;
	SIM_ADD_SHUTTLE : INT := 100;
	SIM_POWER_OFF : INT := 200;
	SIM_INIT_END : INT := 300;
END_VAR
(**)
VAR
	step : INT;
	fbPowerOn : MC_BR_AsmPowerOn_AcpTrak;
	fbPowerOff : MC_BR_AsmPowerOff_AcpTrak;
	fbAddShuttle : MC_BR_SecAddShuttle_AcpTrak;
	shuttlePosition : ARRAY[1..COUNT_OF_SIM_SHUTTLE] OF LREAL;
	loop : USINT;
END_VAR
```

#### Main.st
```iecst
PROGRAM _INIT
	fbPowerOff.Assembly := ADR(gAsmMain);
	fbPowerOn.Assembly := ADR(gAsmMain);
	fbAddShuttle.Sector := ADR(SectorTrackAll);

	FOR loop := 1 TO COUNT_OF_SIM_SHUTTLE BY 1 DO
		shuttlePosition[loop] :=  6.6 + (COUNT_OF_SIM_SHUTTLE * GAP_BETWEEN_OF_SHUTTLE) + ((loop - 1) * GAP_BETWEEN_OF_SHUTTLE);
	END_FOR;

	loop := 1;
END_PROGRAM

PROGRAM _CYCLIC
	CASE step OF
		SIM_POWER_ON:
			fbPowerOn.Execute 		:= TRUE;

			IF fbPowerOn.Done = TRUE THEN
				fbPowerOn.Execute 	:= FALSE;
				step 				:= SIM_ADD_SHUTTLE;
			END_IF

			fbPowerOn();

		SIM_ADD_SHUTTLE:
			fbAddShuttle.Position 	:= shuttlePosition[loop];
			fbAddShuttle.Execute 	:= TRUE;

			IF fbAddShuttle.Done = TRUE THEN
				fbAddShuttle.Execute:= FALSE;

				IF loop < COUNT_OF_SIM_SHUTTLE THEN
					loop			:= loop + 1;
				ELSE
					step 			:= SIM_POWER_OFF;
				END_IF
			END_IF

			fbAddShuttle();

		SIM_POWER_OFF:
			fbPowerOff.Execute 		:= TRUE;

			IF fbPowerOff.Done = TRUE THEN
				fbPowerOff.Execute 	:= FALSE;
				step 				:= SIM_INIT_END;
			END_IF

			fbPowerOff();

		300:

	END_CASE;
END_PROGRAM
```

### Program Logical/Source/Utility/AxisCon (IEC)

#### Variables.var
```iecst
VAR
	MpAxis : ARRAY[0..4] OF MpAxisBasic;
	MpAxisPar : ARRAY[0..4] OF MpAxisBasicParType;
END_VAR
(**)
VAR CONSTANT
	AXIS_MAIN : USINT := 0;
	AXIS01 : USINT := 1;
	AXIS02 : USINT := 2;
	AXIS03 : USINT := 3;
	AXIS04 : USINT := 4;
END_VAR
(**)
VAR
	i : USINT;
END_VAR
```

#### Main.st
```iecst
PROGRAM _INIT

	MpAxis[AXIS_MAIN].MpLink		:= ADR(gAxisMain);
	MpAxis[AXIS_MAIN].Parameters	:= ADR(MpAxisPar[AXIS_MAIN]);
	MpAxis[AXIS_MAIN].Enable		:= TRUE;

	MpAxis[AXIS01].MpLink			:= ADR(gAxis01);
	MpAxis[AXIS01].Parameters		:= ADR(MpAxisPar[AXIS01]);
	MpAxis[AXIS01].Enable			:= TRUE;

	MpAxis[AXIS02].MpLink			:= ADR(gAxis02);
	MpAxis[AXIS02].Parameters		:= ADR(MpAxisPar[AXIS02]);
	MpAxis[AXIS02].Enable			:= TRUE;

	MpAxis[AXIS03].MpLink			:= ADR(gAxis03);
	MpAxis[AXIS03].Parameters		:= ADR(MpAxisPar[AXIS03]);
	MpAxis[AXIS03].Enable			:= TRUE;

	MpAxis[AXIS04].MpLink			:= ADR(gAxis04);
	MpAxis[AXIS04].Parameters		:= ADR(MpAxisPar[AXIS04]);
	MpAxis[AXIS04].Enable			:= TRUE;

END_PROGRAM

PROGRAM _CYCLIC

	FOR i := 0 TO AXIS04 DO
		MpAxis[i]();
	END_FOR;

	IF MpAxis[AXIS_MAIN].Info.ReadyToPowerOn THEN
		MpAxis[AXIS_MAIN].Power	:= TRUE;
	END_IF

END_PROGRAM

PROGRAM _EXIT

	FOR i := 0 TO AXIS04 DO
		MpAxis[i].Enable	:= FALSE;
	END_FOR;

END_PROGRAM
```

### Data object Logical/Source/Utility/AcpParTab (Apt)

#### AcpParTab.apt - ACOPOS Parameter table
```
AcoposParameterTable:
  Root Parameters:
    10 = 33 (Name=R_BLEEDER_EXT, Unit=Ohm)  // Bleeder: External: Resistance
    11 = 637 (Name=TEMP_MAX_BLEEDER_EXT, Unit=캜)  // Bleeder: External: Limit temperature
    12 = 0.9395 (Name=RTH_BLEEDER_AMB_EXT, Unit=K/W)  // Bleeder: External: Thermal resistance
    13 = 40.68 (Name=CTH_BLEEDER_EXT, Unit=Ws/K)  // Bleeder: External: Thermal capacity
```

### Program Logical/Source/Utility/TrakDesign (IEC, version 5.14.0) - trak support: assembly design

#### Init.st - _INIT - set application specific parameter
```iecst
//////////////////////////////////////////////////////////////////////////////////////////////////////////////////////////////
//
// Copyright B&R Industrial Automation GmbH
// Author    B&R
// Created   Feb 1, 2018
//
// trak assembly design support task (optional)
// TC#1 => mandatory to be attached to mappMotion task class
//
// * calculates/estimates the assembly power consumption
// * calculates/estimates the segment power losses
// * analyzes the mechanical situation (does the shuttle stay in the standard-B&R guiding rails?, ist thrust force sufficient?)
// * suitable for use in ARsim (and on real HW)
//
// "TrakDesign" - local interface structure
// "gTrakDesignShuttleOnline" - global interface structure, not mandatory
//
// CAUTION: this task can cause high CPU load on real HW
//
//////////////////////////////////////////////////////////////////////////////////////////////////////////////////////////////

PROGRAM _INIT

	///////////////////////////////////////////////////////////////////////////////////////////////////////////////////////////////////
	// configuration

	// general parameter
	TrakDesign.AssemblyRef			:= ADR(gAsmMain);
	TrakDesign.AssemblyName			:= 'gAsmMain';
	TrakDesign.EnableCalc			:= DiagCpuIsSimulated();	//TRUE;
	TrakDesign.CmdReset				:= FALSE;
	TrakDesign.CmdSaveReport		:= FALSE;
	TrakDesign.CmdRecordToolData	:= FALSE;

	TrakDesign.ParaShuttleType		:= SA102_50N;			//SA201_100D
	TrakDesign.ParaTempAmbient		:= 25;

	//	TrakDesign.ParaMechShuttleIx	:= 1;
	TrakDesign.ParaFileDevice		:= 'SvgData';
	TrakDesign.ParaFileNameReport	:= 'TrakDesignReport.csv';
	TrakDesign.ParaFileNameToolData	:= 'TrakDesignToolData.dat';
	TrakDesign.ParaFileCsvStyle		:= 0;
	TrakDesign.ParaToolDataPrescale	:= 10;

	// shuttle payload parameter
	// carrier
	TrakDesign.Carrier.ParaMass					:= 1.2;			// [kg]
	TrakDesign.Carrier.ParaMassCenterX			:= 0.0;			// [m]
	TrakDesign.Carrier.ParaMassCenterY			:= 0.0;			// [m]
	TrakDesign.Carrier.ParaMassCenterZ			:= 0.0;			// [m]
	TrakDesign.Carrier.ParaMassInertiaZZ		:= 0.0;			// [kg m^2]
	// product
	TrakDesign.Payload[1].ParaName				:= 'no product on carrier';
	TrakDesign.Payload[1].ParaMass				:= 0.0;			// [kg]
	TrakDesign.Payload[1].ParaMassCenterX		:= 0.0;			// [m]
	TrakDesign.Payload[1].ParaMassCenterY		:= 0.0;			// [m]
	TrakDesign.Payload[1].ParaMassCenterZ		:= 0.0;			// [m]
	TrakDesign.Payload[1].ParaMassInertiaZZ		:= 0.0;			// [kg m^2]
	// external friction/force
	TrakDesign.Payload[1].ParaExtFrictionX		:= 0.0;			// [N]
	TrakDesign.Payload[1].ParaExtFrictionVelX	:= 0.0;			// [N/(m/s)]
	TrakDesign.Payload[1].ParaExtForceX			:= 0.0;			// [N]
	TrakDesign.Payload[1].ParaExtForceY			:= 0.0;			// [N]
	TrakDesign.Payload[1].ParaExtForceZ			:= 0.0;			// [N]
	TrakDesign.Payload[1].ParaExtForceAppPointX	:= 0.0;			// [m]
	TrakDesign.Payload[1].ParaExtForceAppPointY	:= 0.0;			// [m]
	TrakDesign.Payload[1].ParaExtForceAppPointZ	:= 0.0;			// [m]

	FOR i:=1 TO TRAK_MAX_SHUTTLE DO
		TrakDesign.Shuttle[i].ParaPayloadIx					:= 1;
		TrakDesign.Shuttle[i].ParaAutoPayload				:= 0;
		//		TrakDesign.Shuttle[i].ParaInitialOrientationFlip	:= 1;
	END_FOR

	// electrical segment assembly
	TrakDesign.Segment[1].ParaName 	:= 'Seg_A_1';		TrakDesign.Segment[1].ParaType := TYPE_BB;		TrakDesign.Segment[1].ParaIxCable := 1;
	TrakDesign.Segment[2].ParaName 	:= 'Seg_A_2';		TrakDesign.Segment[2].ParaType := TYPE_BA;		TrakDesign.Segment[2].ParaIxCable := 1;
	TrakDesign.Segment[3].ParaName 	:= 'Seg_A_3';		TrakDesign.Segment[3].ParaType := TYPE_AA;		TrakDesign.Segment[3].ParaIxCable := 2;
	TrakDesign.Segment[4].ParaName 	:= 'Seg_A_4';		TrakDesign.Segment[4].ParaType := TYPE_AA;		TrakDesign.Segment[4].ParaIxCable := 2;
	TrakDesign.Segment[5].ParaName 	:= 'Seg_A_5';		TrakDesign.Segment[5].ParaType := TYPE_AA;		TrakDesign.Segment[5].ParaIxCable := 2;
	TrakDesign.Segment[6].ParaName 	:= 'Seg_A_6';		TrakDesign.Segment[6].ParaType := TYPE_AA;		TrakDesign.Segment[6].ParaIxCable := 2;
	TrakDesign.Segment[7].ParaName 	:= 'Seg_A_7';		TrakDesign.Segment[7].ParaType := TYPE_AA;		TrakDesign.Segment[7].ParaIxCable := 3;
	TrakDesign.Segment[8].ParaName 	:= 'Seg_A_8';		TrakDesign.Segment[8].ParaType := TYPE_AB;		TrakDesign.Segment[8].ParaIxCable := 3;
	TrakDesign.Segment[9].ParaName 	:= 'Seg_A_9';		TrakDesign.Segment[9].ParaType := TYPE_BB;		TrakDesign.Segment[9].ParaIxCable := 3;
	TrakDesign.Segment[10].ParaName := 'Seg_A_10';		TrakDesign.Segment[10].ParaType := TYPE_BA;		TrakDesign.Segment[10].ParaIxCable := 3;
	TrakDesign.Segment[11].ParaName := 'Seg_A_11';		TrakDesign.Segment[11].ParaType := TYPE_AA;		TrakDesign.Segment[11].ParaIxCable := 4;
	TrakDesign.Segment[12].ParaName := 'Seg_A_12';		TrakDesign.Segment[12].ParaType := TYPE_AA;		TrakDesign.Segment[12].ParaIxCable := 4;
	TrakDesign.Segment[13].ParaName := 'Seg_A_13';		TrakDesign.Segment[13].ParaType := TYPE_AB;		TrakDesign.Segment[13].ParaIxCable := 4;
	TrakDesign.Segment[14].ParaName := 'Seg_A_14';		TrakDesign.Segment[14].ParaType := TYPE_BB;		TrakDesign.Segment[14].ParaIxCable := 4;
	TrakDesign.Segment[15].ParaName := 'Seg_A_15';		TrakDesign.Segment[15].ParaType := TYPE_BA;		TrakDesign.Segment[15].ParaIxCable := 4;
	TrakDesign.Segment[16].ParaName := 'Seg_A_16';		TrakDesign.Segment[16].ParaType := TYPE_AA;		TrakDesign.Segment[16].ParaIxCable := 5;
	TrakDesign.Segment[17].ParaName := 'Seg_A_17';		TrakDesign.Segment[17].ParaType := TYPE_AA;		TrakDesign.Segment[17].ParaIxCable := 5;
	TrakDesign.Segment[18].ParaName := 'Seg_A_18';		TrakDesign.Segment[18].ParaType := TYPE_AA;		TrakDesign.Segment[18].ParaIxCable := 5;
	TrakDesign.Segment[19].ParaName := 'Seg_A_19';		TrakDesign.Segment[19].ParaType := TYPE_AA;		TrakDesign.Segment[19].ParaIxCable := 5;
	TrakDesign.Segment[20].ParaName := 'Seg_A_20';		TrakDesign.Segment[20].ParaType := TYPE_AA;		TrakDesign.Segment[20].ParaIxCable := 6;
	TrakDesign.Segment[21].ParaName := 'Seg_A_21';		TrakDesign.Segment[21].ParaType := TYPE_AB;		TrakDesign.Segment[21].ParaIxCable := 6;
	TrakDesign.Segment[22].ParaName := 'Seg_A_22';		TrakDesign.Segment[22].ParaType := TYPE_BB;		TrakDesign.Segment[22].ParaIxCable := 6;
	TrakDesign.Segment[23].ParaName := 'Seg_A_23';		TrakDesign.Segment[23].ParaType := TYPE_BA;		TrakDesign.Segment[22].ParaIxCable := 7;
	TrakDesign.Segment[24].ParaName := 'Seg_A_24';		TrakDesign.Segment[24].ParaType := TYPE_AA;		TrakDesign.Segment[22].ParaIxCable := 7;
	TrakDesign.Segment[25].ParaName := 'Seg_A_25';		TrakDesign.Segment[25].ParaType := TYPE_AA;		TrakDesign.Segment[22].ParaIxCable := 7;
	TrakDesign.Segment[26].ParaName := 'Seg_A_26';		TrakDesign.Segment[26].ParaType := TYPE_AB;		TrakDesign.Segment[22].ParaIxCable := 1;

	// power cable assembly
	TrakDesign.Cable[1].ParaLength := 10.0;						TrakDesign.Cable[1].ParaIxSupply := 1;
	TrakDesign.Cable[2].ParaLength := 10.0;						TrakDesign.Cable[2].ParaIxSupply := 2;
	TrakDesign.Cable[3].ParaLength := 10.0;						TrakDesign.Cable[3].ParaIxSupply := 3;
	TrakDesign.Cable[4].ParaLength := 10.0;						TrakDesign.Cable[4].ParaIxSupply := 4;
	TrakDesign.Cable[5].ParaLength := 5.0;						TrakDesign.Cable[5].ParaIxSupply := 5;
	TrakDesign.Cable[6].ParaLength := 5.0;						TrakDesign.Cable[6].ParaIxSupply := 6;
	TrakDesign.Cable[7].ParaLength := 5.0;						TrakDesign.Cable[6].ParaIxSupply := 7;
	// power supply assembly
	TrakDesign.Supply[1].ParaName := 'gAxis01';					TrakDesign.Supply[1].ParaType := BC032;			TrakDesign.Supply[1].ParaIxSupplyParallel := 1;
	TrakDesign.Supply[2].ParaName := 'gAxis01';					TrakDesign.Supply[2].ParaType := BC032;			TrakDesign.Supply[2].ParaIxSupplyParallel := 2;
	TrakDesign.Supply[3].ParaName := 'gAxis02';					TrakDesign.Supply[3].ParaType := BC032;			TrakDesign.Supply[3].ParaIxSupplyParallel := 3;
	TrakDesign.Supply[4].ParaName := 'gAxis02';					TrakDesign.Supply[4].ParaType := BC032;			TrakDesign.Supply[4].ParaIxSupplyParallel := 4;
	TrakDesign.Supply[5].ParaName := 'gAxis03';					TrakDesign.Supply[5].ParaType := BC032;			TrakDesign.Supply[5].ParaIxSupplyParallel := 5;
	TrakDesign.Supply[6].ParaName := 'gAxis03';					TrakDesign.Supply[6].ParaType := BC032;			TrakDesign.Supply[6].ParaIxSupplyParallel := 6;
	TrakDesign.Supply[7].ParaName := 'gAxis04';					TrakDesign.Supply[7].ParaType := BC032;			TrakDesign.Supply[7].ParaIxSupplyParallel := 7;

	ExpertReport := TRUE;
	CreateFileHistory := TRUE;

	Action_INIT;

END_PROGRAM
```

- Main.st (not readable text: treated as protected, skipped)
